// IndraMotionMlc1/Application/CheckBounds
(*
General Header
----------------------------------------------------------------------------------------------
Short description      : Function to check access to array within valid bounds.
                         After inserting/removing this function, no online-change will be possible! A complete download will be necessary!
Version                : 14.1.0.0
Author                 : DC-IA/EAM3 (MD)
Date                   : 2015-01-12
Company                : Bosch Rexroth AG
Target                 : IndraLogic XLC/MLC
Functional description : This function will be called implicitly before the read/write access
                         to arrays takes places.
                         The index of the subsequent array accesses is checked for valid
                         limits.
                         In case of invalid access, an error is entered in the diagnostic
                         logbook and the application is stopped due to an access violation to
                         avoid machine damage.
                         In this case, check the callstack (menu Debug/Callstack) and modify
                         the faulty logic. 
Handling specials      : This function increases the cycle time of all IEC-tasks using array
                         accesses. 
                         The increase depends on the number of the read/write accesses to
                         arrays.
                         After inserting/removing this function, no online-change will be possible! 
                         A complete download will be necessary!
						 This is an exemplary implementation of the function. 
                         The implementation has to be adjusted to your application/machine.
						 Per default, the PLC-Task will generate an access violation which leads to
                         an application stop and a F5-error with error reaction respectively.
                         Please verify whether this default behaviour can damage your machine 
                         or lead to a complex recommissioning. 
                         In this case, adapt the error reaction to your application.
						 
                         If your application isn't too time-critical, you should leave this function 
						 while commissioning the machine and production in your application.  
                         If you remove this funciton, ensure that your code is faultless.
                         
                         Do not modify the declaration of this function! 
                         Do not change the attributes above the function header!
----------------------------------------------------------------------------------------------
*)
{attribute 'check_bounds'}
{attribute 'no_check'}
{attribute 'signature_flag' := '1073741824'}
FUNCTION CheckBounds : DINT
VAR_INPUT
	index, lower, upper: DINT;
END_VAR
VAR
	{attribute 'hide'}
	bByte: BYTE;
	ptNull: POINTER TO BYTE :=0;
	errstr: STRING;
	
END_VAR

(*************************************************************
This function was generated by the 'check array access'
option of the controllers 'properties' dialog box.
If you delete this comment, the 'check array access' option
of the controllers 'properties' dialog box will be removed.
**************************************************************)
    (**************************************************************************************************)
    (* The implementation has to be adjusted to your application/machine.                             *)
    (* This is an exemplary implementation of the function.                                           *)
    (* Per default, an access violation is generated to avoid machine damage                          *)
    (* Check the Call Stack (menu Debug/Callstack) and modify the faulty logic!                       *)
    (**************************************************************************************************)

IF  index < lower THEN 
	errstr:= 'CheckBounds: Lower arrayindex ';
	errstr:=CONCAT(STR1:=errstr  , STR2:= DINT_TO_STRING(lower));
	errstr:=CONCAT(STR1:=errstr  , STR2:= ' underrunned by ');
	errstr:=CONCAT(STR1:=errstr  , STR2:= DINT_TO_STRING(index));
//  This pragma may be removed: 
	{info 'CheckBounds: Please implement your own error reaction below'}
//  EXAMPLE 1 (default): 
//  Set a F0-Error into the diagnostic- and error memory
//  Triggering an access violation --> Application will be stopped and leads to a F5-Error

  ML_SetDiagEntry(
	Severity:= E_LOG_SEVERITY.ERROR, 
	Class:= E_LOG_CLASS.CLASS_0, 
	Facility:= E_LOG_FACILITY.USER, 
	Code:= 0, 
	Text:= ADR(errstr));

	bByte:=ptNull^;(*triggering an access violation *)

// EXAMPLE 2:
// Limit the faulty index to the lower index 
//     -> no memory will be overwritten
//     -> Keep PLC-task and motion running
// Set a E0-Warning into the diagnostic- and error memory
// NOTE: There is still an implementation error in your application code!

//  ML_SetDiagEntry(
//	Severity:= E_LOG_SEVERITY.WARNING, 
//	Class:= E_LOG_CLASS.CLASS_0, 
//	Facility:= E_LOG_FACILITY.USER, 
//	Code:= 0, 
//	Text:= ADR(errstr));
// 
//	CheckBounds := lower; //access to the lower index only 
//  return;
	
ELSIF  index > upper THEN
	errstr:= 'CheckBounds: Higher arrayindex ';
	errstr:=CONCAT(STR1:=errstr  , STR2:= DINT_TO_STRING(upper));
	errstr:=CONCAT(STR1:=errstr  , STR2:= ' overrunned by ');
	errstr:=CONCAT(STR1:=errstr  , STR2:= DINT_TO_STRING(index));

//  this pragma may be removed: 
	{info 'CheckBounds: Please implement your own error reaction below'}
//  example 1 (default): 
//  set a F0-Error into the diagnostic- and error memory
//  triggering an access violation --> Application will be stopped and leads to a F5-Error

  ML_SetDiagEntry(
	Severity:= E_LOG_SEVERITY.ERROR, 
	Class:= E_LOG_CLASS.CLASS_0, 
	Facility:= E_LOG_FACILITY.USER, 
	Code:= 0, 
	Text:= ADR(errstr));

	bByte:=ptNull^;(*triggering an access violation *)

//example 2:
// Limit the faulty index to the upper index 
//     -> no memory will be overwritten
//     -> Keep PLC-task and motion running
// Set a E0-Warning into the diagnostic- and error memory
// NOTE: There is still an implementation error in your application code!

//  ML_SetDiagEntry(
//	Severity:= E_LOG_SEVERITY.WARNING, 
//	Class:= E_LOG_CLASS.CLASS_0, 
//	Facility:= E_LOG_FACILITY.USER, 
//	Code:= 0, 
//	Text:= ADR(errstr));
// 
//	CheckBounds := upper; //access to the upper index only 
//  return;

ELSE // access to array is ok  
	CheckBounds := index;
END_IF

END_FUNCTION

// IndraMotionMlc1/Application/POUs/Useless/MotionProg
PROGRAM MotionProg
VAR
	b_enable_1: BOOL;
	MC_Power_0: MC_POWER;
	b_enable_on_1: BOOL;
	b_move_1: BOOL;
	MC_MoveVelocity_0: MC_MoveVelocity;
	vel: REAL;
	b_enable_2: BOOL;
	MC_Power_1: MC_POWER;
	b_enable_on_2: BOOL;
	b_move_2: BOOL;
	MC_MoveVelocity_1: MC_MoveVelocity;
	b_enable_3: BOOL;
	MC_Power_2: MC_POWER;
	b_enable_on_3: BOOL;
	b_move_3: BOOL;
	MC_MoveVelocity_2: MC_MoveVelocity;
	b_power: BOOL;
	b_vel_az1: BOOL;
	b_enable_az1: BOOL;
	b_enable_az2: BOOL;
	b_torque_az2: BOOL;
	b_torque_on_2: BOOL;
	MC_torque_az2: MC_TorqueControl;
	b_enable_el_1: BOOL;
	b_move_el_1: BOOL;
	b_torque_az1: BOOL;
	MC_torque_az1: MC_TorqueControl;
	b_torque_on_1: BOOL;
	b_vel_2: BOOL;
END_VAR

motionprog.P_MOTION();

ACTION P_MOTION:
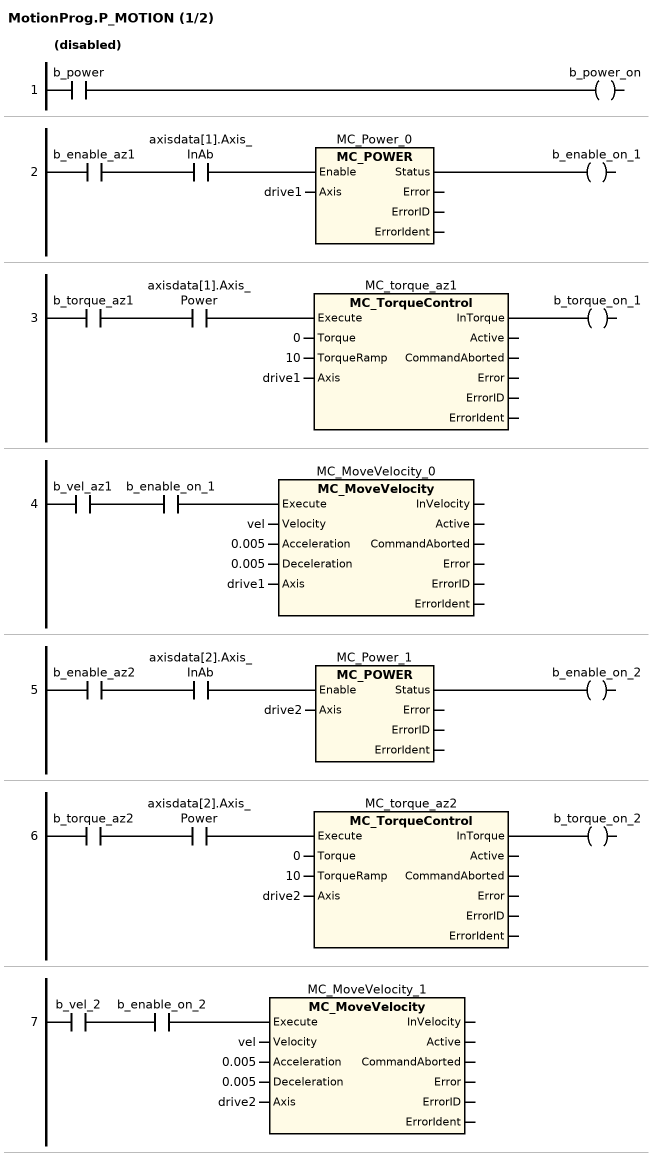
// NETWORK 1 (disabled)
// b_power_on := b_power;

// NETWORK 2
MC_Power_0(Enable := b_enable_az1 AND axisdata[1].Axis_InAb, Axis := drive1); // MC_POWER
b_enable_on_1 := MC_Power_0.Status;

// NETWORK 3
MC_torque_az1(
    Execute := b_torque_az1 AND axisdata[1].Axis_Power,
    Torque := 0,
    TorqueRamp := 10,
    Axis := drive1); // MC_TorqueControl
b_torque_on_1 := MC_torque_az1.InTorque;

// NETWORK 4
MC_MoveVelocity_0(
    Execute := b_vel_az1 AND b_enable_on_1,
    Velocity := vel,
    Acceleration := 0.005,
    Deceleration := 0.005,
    Axis := drive1); // MC_MoveVelocity

// NETWORK 5
MC_Power_1(Enable := b_enable_az2 AND axisdata[2].Axis_InAb, Axis := drive2); // MC_POWER
b_enable_on_2 := MC_Power_1.Status;

// NETWORK 6
MC_torque_az2(
    Execute := b_torque_az2 AND axisdata[2].Axis_Power,
    Torque := 0,
    TorqueRamp := 10,
    Axis := drive2); // MC_TorqueControl
b_torque_on_2 := MC_torque_az2.InTorque;

// NETWORK 7
MC_MoveVelocity_1(
    Execute := b_vel_2 AND b_enable_on_2,
    Velocity := vel,
    Acceleration := 0.005,
    Deceleration := 0.005,
    Axis := drive2); // MC_MoveVelocity

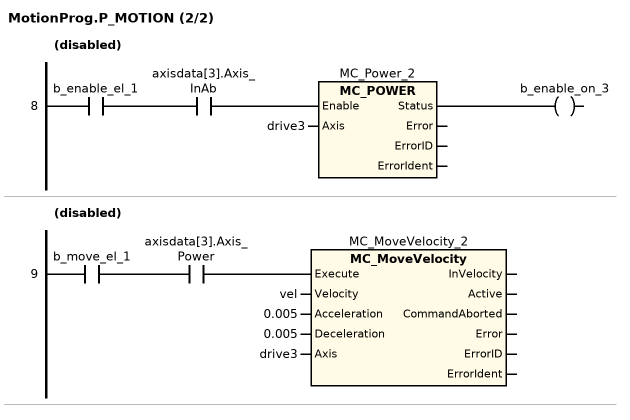
// NETWORK 8 (disabled)
// MC_Power_2(Enable := b_enable_el_1 AND axisdata[3].Axis_InAb, Axis := drive3); // MC_POWER
// b_enable_on_3 := MC_Power_2.Status;

// NETWORK 9 (disabled)
// MC_MoveVelocity_2(
//     Execute := b_move_el_1 AND axisdata[3].Axis_Power,
//     Velocity := vel,
//     Acceleration := 0.005,
//     Deceleration := 0.005,
//     Axis := drive3); // MC_MoveVelocity
END_ACTION

END_PROGRAM

// IndraMotionMlc1/Application/POUs/Panel Function/P_LED
(*
This progrom is bulit for lighting the led in the panelbox which describe the limit.
1)If the angle is reach the limit value,we use the Function Block MB_WriteParameter to setting 
special value to the parameter FP_P_0_0304 of the relative drive.so that the led will be lighted.
2)Besides,when the position of azimuth axis is at the zone,60 degrees nearby the limit,the led of azimuth will flicker every 2 seconds.
Similar with azimuth,the elevation LED will flicker at the 5-degrees-zone nearby limit,and the FeedIndexer LED will flicker at the 30-degrees-zone nearby limit.
*)
PROGRAM P_LED
VAR
(*the definition of Blink function blocks*)
	fb_blink_LED_az: BLINK;
	fb_blink_write_az: BLINK;
	fb_blink_LED_el: BLINK;
	fb_blink_write_el: BLINK;
	fb_blink_LED_FI: BLINK;
	fb_blink_write_FI: BLINK;
	t_LED_az: TIME;
	t_LED_el: TIME;
	t_LED_FI: TIME;
	b_LED_az: BOOL;
	b_LED_el: BOOL;
	b_LED_FI: BOOL;
(*the definition of function blocks for Writing p304 Parameter*)
	fb_write_p304_d2: MB_WriteParameter;(*the I/O of azimuth LED is on drive2*)
	fb_write_p304_d4: MB_WriteParameter;(*the I/O of elevation LED is on drive4*)
	fb_write_p304_d5: MB_WriteParameter;(*the I/O of FeedIndexer LED is on drive5*)
(*when the P304 parameter equal to 512,only the 9th on the I/O is set;
when the P304 parameter equal to 1024,only the 10th on the I/O is set;
when the P304 parameter equal to 0,all the I/O is reset;*)
	i_p304_az: INT;
	i_p304_el: INT;
	i_p304_FI: INT;
END_VAR

IF b_local_on=TRUE THEN
	b_local_led:=TRUE;
ELSE
	b_local_led:=FALSE;
END_IF

IF b_remote_on=TRUE THEN
	b_remote_led:=TRUE;
ELSE
	b_remote_led:=FALSE;
END_IF

IF b_ESTOP_door=TRUE THEN
	b_estop_led :=TRUE;
ELSE
	b_estop_led :=FALSE;
END_IF

   IF master_status.4 =FALSE THEN
	   b_normal_led:=TRUE;
	   b_error_led:=FALSE;
   ELSE
   	   b_normal_led:=FALSE;
	   b_error_led:=TRUE;
   END_IF


(*
IF b_local_on=TRUE THEN
(*<<<<<<<<<<<<<<<<<<<<<<<<<<<<<<<<LED Of azimuth>>>>>>>>>>>>>>>>>>>>>>>>>>>>>>>>>*)
	IF r_pos_az>=0 AND r_pos_az<=180 THEN
		i_p304_az:=0;
	ELSIF r_pos_az>180 AND r_pos_az<358.5 THEN
		t_LED_az:=T#2.2s;
		IF b_LED_az= TRUE THEN
			i_p304_az:=0;
		ELSE
			i_p304_az:=512;
		END_IF
	ELSIF r_pos_az>=358.5 THEN
		i_p304_az:=512;
	ELSIF r_pos_az<0 AND r_pos_az>-178.5 THEN
		t_LED_az:=T#2.2s;
		IF b_LED_az= TRUE THEN
			i_p304_az:=0;
		ELSE
			i_p304_az:=1024;
		END_IF
	ELSIF r_pos_az<=-178.5 THEN
		i_p304_az:=1024;
	END_IF
(*<<<<<<<<<<<<<<<<<<<<<<<<<<<<<<<<LED Of elevation>>>>>>>>>>>>>>>>>>>>>>>>>>>>>>>>>*)
	IF r_pos_el>=25 AND r_pos_el<=80 THEN
		i_p304_el:=0;
	ELSIF r_pos_el>80 AND r_pos_el<=90.1 THEN
		t_LED_el:=T#2.2s;
		IF b_LED_el= TRUE THEN
			i_p304_el:=0;
		ELSE
			i_p304_el:=512;
		END_IF
	ELSIF r_pos_el>90.1 THEN
		i_p304_el:=512;
	ELSIF r_pos_el>25 AND r_pos_el<=15 THEN
		t_LED_el:=T#2.2s;
		IF b_LED_el= TRUE THEN
			i_p304_el:=0;
		ELSE
			i_p304_el:=1024;
		END_IF
	ELSIF r_pos_el<15 THEN
		i_p304_el:=1024;
	END_IF
(*<<<<<<<<<<<<<<<<<<<<<<<<<<<<<<<<LED Of FeedIndexer>>>>>>>>>>>>>>>>>>>>>>>>>>>>>>>>>*)
	IF r_pos_FI>=-120 AND r_pos_FI<=120 THEN
		i_p304_FI:=0;
	ELSIF r_pos_FI>120 AND r_pos_FI<=178.5 THEN
		t_LED_FI:=T#2.2s;
		IF b_LED_FI= TRUE THEN
			i_p304_FI:=0;
		ELSE
			i_p304_FI:=512;
		END_IF
	ELSIF r_pos_FI>178.5 THEN
		i_p304_FI:=512;
	ELSIF r_pos_FI<-120 AND r_pos_FI>=-178.5 THEN
		t_LED_FI:=T#2.2s;
		IF b_LED_FI= TRUE THEN
			i_p304_FI:=0;
		ELSE
			i_p304_FI:=1024;
		END_IF
	ELSIF r_pos_FI<-178.5 THEN
		i_p304_FI:=1024;
	END_IF
ELSE
(*if not at local situation,the LED is dark*)
(*For testing LED,write i_p304_az:=1536;i_p304_el:=1536;i_p304_FI:=1536;*)
	i_p304_az:=0;
	i_p304_el:=0;
	i_p304_FI:=0;
END_IF

(*transfer the sub-program A_w_P304 to white value to the parameter FP_P_0_0304*)
P_LED.A_w_P304;*)

ACTION A_w_P304:
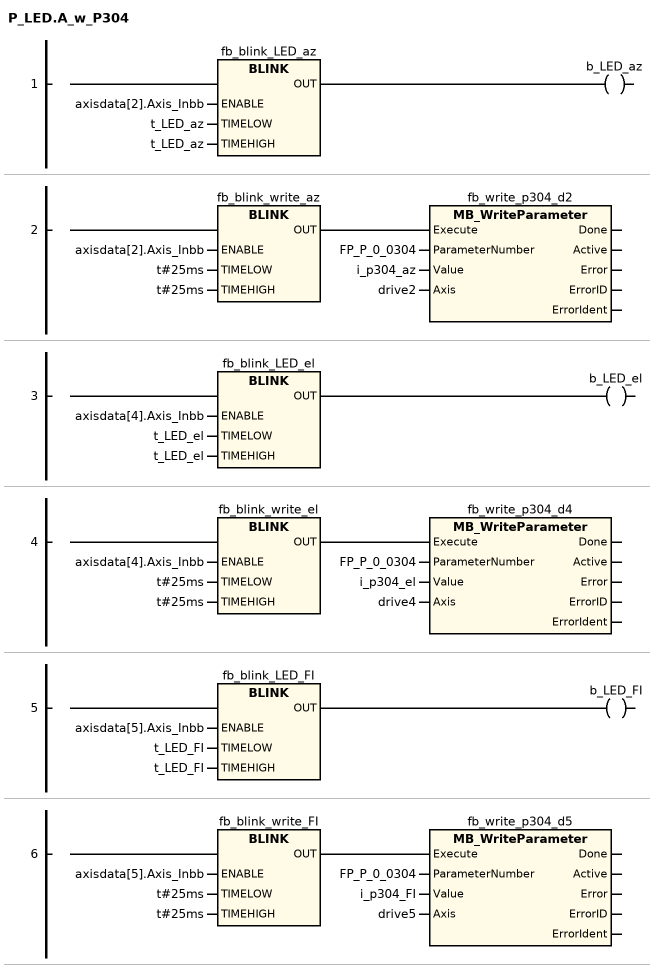
// NETWORK 1
fb_blink_LED_az(ENABLE := axisdata[2].Axis_Inbb, TIMELOW := t_LED_az, TIMEHIGH := t_LED_az); // BLINK
b_LED_az := fb_blink_LED_az.OUT;

// NETWORK 2
fb_blink_write_az(ENABLE := axisdata[2].Axis_Inbb, TIMELOW := t#25ms, TIMEHIGH := t#25ms); // BLINK
fb_write_p304_d2(
    Execute := fb_blink_write_az.OUT,
    ParameterNumber := FP_P_0_0304,
    Value := i_p304_az,
    Axis := drive2); // MB_WriteParameter

// NETWORK 3
fb_blink_LED_el(ENABLE := axisdata[4].Axis_Inbb, TIMELOW := t_LED_el, TIMEHIGH := t_LED_el); // BLINK
b_LED_el := fb_blink_LED_el.OUT;

// NETWORK 4
fb_blink_write_el(ENABLE := axisdata[4].Axis_Inbb, TIMELOW := t#25ms, TIMEHIGH := t#25ms); // BLINK
fb_write_p304_d4(
    Execute := fb_blink_write_el.OUT,
    ParameterNumber := FP_P_0_0304,
    Value := i_p304_el,
    Axis := drive4); // MB_WriteParameter

// NETWORK 5
fb_blink_LED_FI(ENABLE := axisdata[5].Axis_Inbb, TIMELOW := t_LED_FI, TIMEHIGH := t_LED_FI); // BLINK
b_LED_FI := fb_blink_LED_FI.OUT;

// NETWORK 6
fb_blink_write_FI(ENABLE := axisdata[5].Axis_Inbb, TIMELOW := t#25ms, TIMEHIGH := t#25ms); // BLINK
fb_write_p304_d5(
    Execute := fb_blink_write_FI.OUT,
    ParameterNumber := FP_P_0_0304,
    Value := i_p304_FI,
    Axis := drive5); // MB_WriteParameter
END_ACTION

END_PROGRAM

// IndraMotionMlc1/Application/POUs/Panel Function/P_Lock_Panel_TCP
(*This program is bulit for lock the antenna for stow and maintain,and for unlock the antenna.
It mainly contains goto function,the control of AC moter,and the protect for safety*)
PROGRAM P_Lock_Panel_TCP
VAR

(*<<<<<<<<<<<<<<<<<<<the allow for the lock moter>>>>>>>>>>>>>>>>>*)
	b_lock_allow_0: BOOL;
	b_lock_allow_20: BOOL;
(*the definition of rise trigger,The function block R_TRIG detects a rising edge. *)
	rtrig_lock_stow: R_TRIG;
	rtrig_lock_maintain: R_TRIG;
	rtrig_reset_TCP_unlock: R_TRIG;
	rtrig_reset_TCP_lock: R_TRIG;
	rtrig_enable_unlock: R_TRIG;
(*The function block Timer On Delay implements a turn-on delay*)
	ton_stow_0: TON;
	ton_maintain_20: TON;
	ton_reset_lock: TON;
	ton_reset_unlock: TON;
(*the fixed position according to the hole*)
	r_postion_stow: REAL;
	r_position_maintain: REAL;
(*move the elevation to the fixed position*)
	fb_move_AZ_0: MC_MoveAbsolute;
	fb_move_el_20: MC_MoveAbsolute;
	fb_self_reset_stow: R_TRIG;
	fb_ton_self_reset_stow: TON;
	b_lock_allow_21: BOOL;
	fb_self_reset_maintain: R_TRIG;
	fb_ton_self_reset_maintain: TON;
	b_off_stow: R_TRIG;
	b_off_maintain: R_TRIG;
	fb_move_EL_0: MC_MoveAbsolute;
END_VAR

(*<<<<<<<<<<<<<<<<<<<<write the stow and maintain position according to IP>>>>>>>>>>>>>>>>>>>>>>>>>>>>>>>>>>>>*)
(*every antenna maybe has the different stow position and maintain position from the others*)
str_1xx:=RIGHT(str_MLC_ip,3);(*for get the last 3 number of IP in MLC*)
IF str_1xx='101' THEN
	r_postion_stow:=0;
	r_position_maintain:=20.15;
ELSIF str_1xx='102' THEN
	r_postion_stow:=0;
	r_position_maintain:=20.820;
ELSIF str_1xx='103' THEN
	r_postion_stow:=0;
	r_position_maintain:=20.950;
ELSIF str_1xx='104' THEN
	r_postion_stow:=0;
	r_position_maintain:=20.9;
ELSIF str_1xx='105' THEN
	r_postion_stow:=0;
	r_position_maintain:=20.930;
ELSIF str_1xx='106' THEN
	r_postion_stow:=0;
	r_position_maintain:=20.800;
ELSIF str_1xx='107' THEN
	r_postion_stow:=90.00;
	r_position_maintain:=20.850;
ELSIF str_1xx='108' THEN
	r_postion_stow:=90.00;
	r_position_maintain:=21.100;
ELSIF str_1xx='109' THEN
	r_postion_stow:=90.00;
	r_position_maintain:=21.000;
ELSIF str_1xx='110' THEN
	r_postion_stow:=0;
	r_position_maintain:=21.000;
ELSIF str_1xx='111' THEN
	r_postion_stow:=0;
	r_position_maintain:=21.000;
ELSIF str_1xx='112' THEN
	r_postion_stow:=0;
	r_position_maintain:=21.100;
ELSIF str_1xx='113' THEN
	r_postion_stow:=0;
	r_position_maintain:=21.000;
ELSIF str_1xx='114' THEN
	r_postion_stow:=0;
	r_position_maintain:=21.000;
ELSIF str_1xx='115' THEN
	r_postion_stow:=0;
	r_position_maintain:=21.000;
ELSIF str_1xx='116' THEN
	r_postion_stow:=0;
	r_position_maintain:=21.000;
ELSIF str_1xx='117' THEN
	r_postion_stow:=0;
	r_position_maintain:=21.000;
ELSIF str_1xx='118' THEN
	r_postion_stow:=0;
	r_position_maintain:=20.950;
ELSIF str_1xx='119' THEN
	r_postion_stow:=0;
	r_position_maintain:=20.950;
ELSIF str_1xx='120' THEN
	r_postion_stow:=0;
	r_position_maintain:=21.000;
ELSIF str_1xx='121' THEN
	r_postion_stow:=0;
	r_position_maintain:=21.000;
ELSIF str_1xx='122' THEN
	r_postion_stow:=0;
	r_position_maintain:=21.000;
ELSIF str_1xx='123' THEN
	r_postion_stow:=0;
	r_position_maintain:=21.000;
ELSIF str_1xx='124' THEN
	r_postion_stow:=0;
	r_position_maintain:=21.000;
ELSIF str_1xx='125' THEN
	r_postion_stow:=0;
	r_position_maintain:=21.000;
ELSIF str_1xx='126' THEN
	r_postion_stow:=0;
	r_position_maintain:=21.000;
ELSIF str_1xx='127' THEN
	r_postion_stow:=0;
	r_position_maintain:=21.000;
ELSIF str_1xx='128' THEN
	r_postion_stow:=0;
	r_position_maintain:=21.000;
ELSIF str_1xx='129' THEN
	r_postion_stow:=0;
	r_position_maintain:=21.000;
ELSIF str_1xx='130' THEN
	r_postion_stow:=0;
	r_position_maintain:=20.950;
ELSIF str_1xx='131' THEN
	r_postion_stow:=0;
	r_position_maintain:=21.000;
ELSIF str_1xx='132' THEN
	r_postion_stow:=0;
	r_position_maintain:=21.000;
ELSIF str_1xx='133' THEN
	r_postion_stow:=0;
	r_position_maintain:=21.000;
ELSIF str_1xx='134' THEN
	r_postion_stow:=0;
	r_position_maintain:=21.000;
ELSIF str_1xx='135' THEN
	r_postion_stow:=0.00;
	r_position_maintain:=21.000;
ELSIF str_1xx='136' THEN
	r_postion_stow:=0.00;
	r_position_maintain:=21.000;

(*test*)
ELSIF str_1xx='1.1' THEN
	r_postion_stow:=0.00;
	r_position_maintain:=20.9;
ELSE
	r_postion_stow:=0;
	r_position_maintain:=11;
END_IF
(*<<<<<<<<<<<<<<<<<<<<<<<<<<<<<<<<if the elevation position is nearby the fixed value,then allow the lock action>>>>>>>>>>>>>>>>>>>>>>>>>>>>>>>>>>>>>>>>>>>>>>>>>>>*)
IF ABS(axisdata[1].rActualPosition_i-0)<0.01 THEN
	b_lock_allow_0:=TRUE;
ELSE
	b_lock_allow_0:=FALSE;
END_IF

IF b_stow_pin_limit_lock = FALSE AND ABS(axisdata[1].rActualPosition_i-r_postion_stow)< 0.1 THEN
	b_stow_lock:=TRUE;
ELSE
	b_stow_lock:=FALSE;
END_IF;

P_Lock_Panel_TCP.A_LOCK();

ACTION A_LOCK:
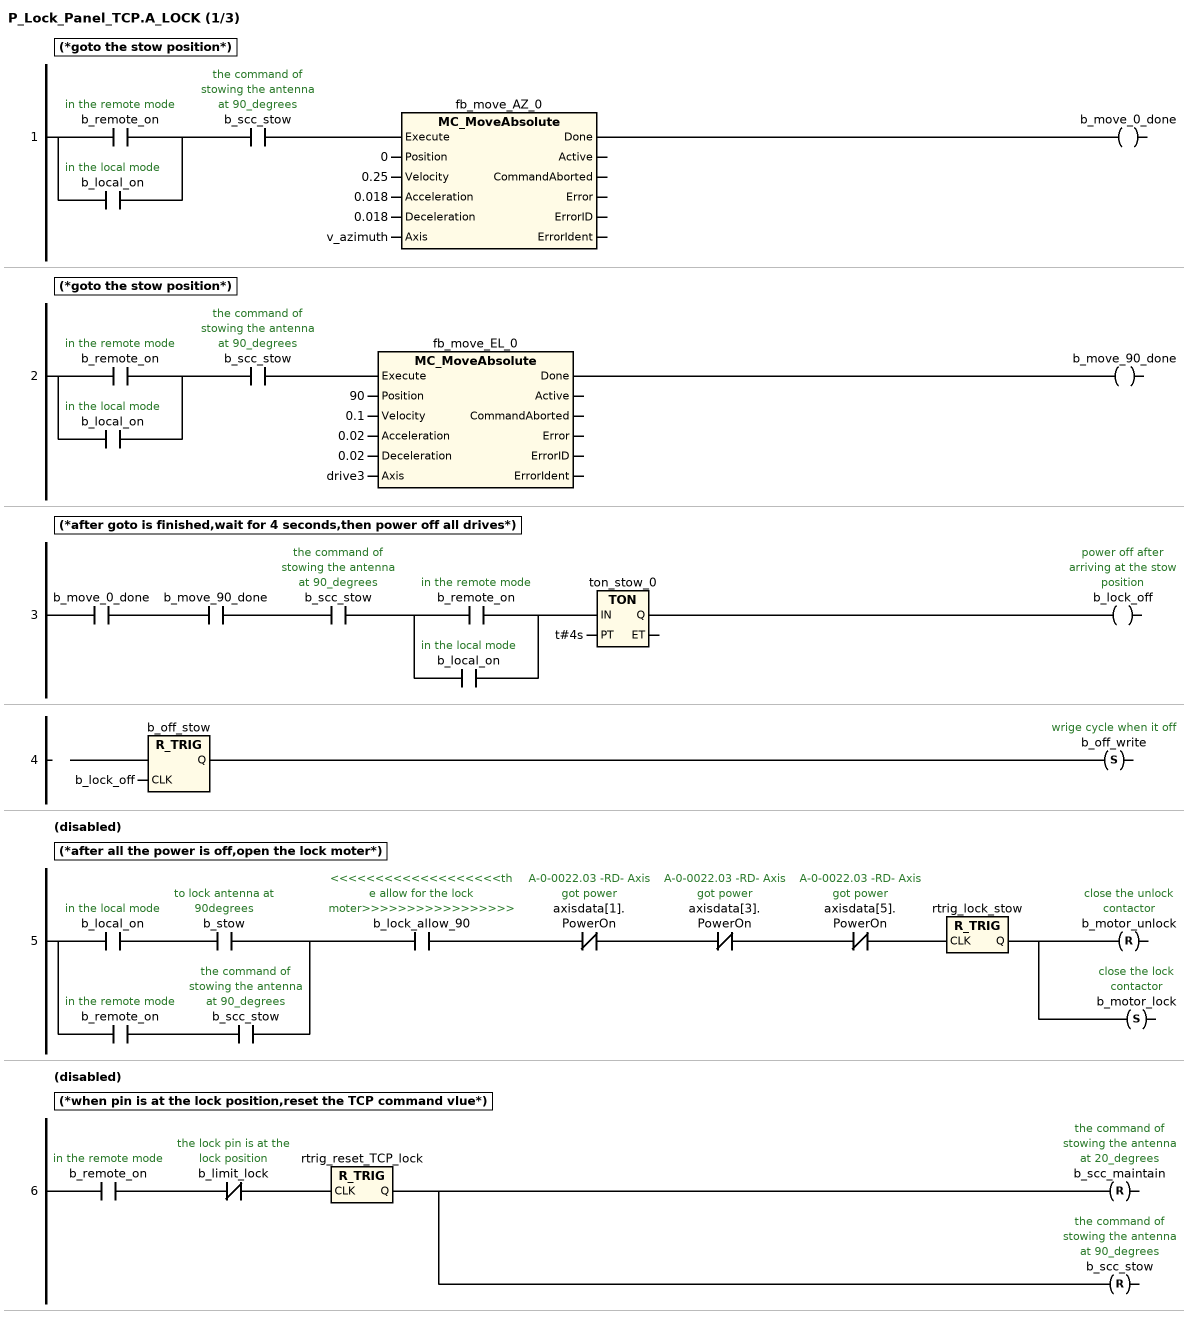
// NETWORK 1
//   fb_move_AZ_0: move the elevation to the fixed position
//   b_remote_on: in the remote mode
//   b_local_on: in the local mode
//   b_scc_stow: the command of stowing the antenna at 90_degrees
//   v_azimuth: Virtual axis "v_elevation" with axis number 8
// label: (*goto the stow position*)
fb_move_AZ_0(
    Execute := (b_remote_on OR b_local_on) AND b_scc_stow,
    Position := 0,
    Velocity := 0.25,
    Acceleration := 0.018,
    Deceleration := 0.018,
    Axis := v_azimuth); // MC_MoveAbsolute
b_move_0_done := fb_move_AZ_0.Done;

// NETWORK 2
//   fb_move_EL_0: move the elevation to the fixed position
//   b_remote_on: in the remote mode
//   b_local_on: in the local mode
//   b_scc_stow: the command of stowing the antenna at 90_degrees
//   drive3: Virtual axis "v_elevation" with axis number 8
// label: (*goto the stow position*)
fb_move_EL_0(
    Execute := (b_remote_on OR b_local_on) AND b_scc_stow,
    Position := 90,
    Velocity := 0.1,
    Acceleration := 0.02,
    Deceleration := 0.02,
    Axis := drive3); // MC_MoveAbsolute
b_move_90_done := fb_move_EL_0.Done;

// NETWORK 3
//   ton_stow_0: The function block Timer On Delay implements a turn-on delay
//   b_scc_stow: the command of stowing the antenna at 90_degrees
//   b_remote_on: in the remote mode
//   b_local_on: in the local mode
//   b_lock_off: power off after arriving at the stow position
// label: (*after goto is finished,wait for 4 seconds,then power off all drives*)
ton_stow_0(IN := b_move_0_done AND b_move_90_done AND b_scc_stow AND (b_remote_on OR b_local_on), PT := t#4s); // TON
b_lock_off := ton_stow_0.Q;

// NETWORK 4
//   b_lock_off: power off after arriving at the stow position
//   b_off_write: wrige cycle when it off
b_off_stow(CLK := b_lock_off); // R_TRIG
b_off_write S= b_off_stow.Q;

// NETWORK 5 (disabled)
//   rtrig_lock_stow: the definition of rise trigger,The function block R_TRIG detects a rising edge.
//   b_local_on: in the local mode
//   b_stow: to lock antenna at 90degrees
//   b_remote_on: in the remote mode
//   b_scc_stow: the command of stowing the antenna at 90_degrees
//   b_lock_allow_90: <<<<<<<<<<<<<<<<<<<the allow for the lock moter>>>>>>>>>>>>>>>>>
//   axisdata[1].PowerOn: A-0-0022.03 -RD- Axis got power
//   axisdata[3].PowerOn: A-0-0022.03 -RD- Axis got power
//   axisdata[5].PowerOn: A-0-0022.03 -RD- Axis got power
//   b_motor_unlock: close the unlock contactor
//   b_motor_lock: close the lock contactor
// label: (*after all the power is off,open the lock moter*)
// rtrig_lock_stow(CLK := (b_local_on AND b_stow OR b_remote_on AND b_scc_stow) AND b_lock_allow_90 AND NOT axisdata[1].PowerOn AND NOT axisdata[3].PowerOn AND NOT axisdata[5].PowerOn); // R_TRIG
// b_motor_unlock R= rtrig_lock_stow.Q;
// b_motor_lock S= rtrig_lock_stow.Q;

// NETWORK 6 (disabled)
//   b_remote_on: in the remote mode
//   b_limit_lock: the lock pin is at the lock position
//   b_scc_maintain: the command of stowing the antenna at 20_degrees
//   b_scc_stow: the command of stowing the antenna at 90_degrees
// label: (*when pin is at the lock position,reset the TCP command vlue*)
// rtrig_reset_TCP_lock(CLK := b_remote_on AND NOT b_limit_lock); // R_TRIG
// b_scc_maintain R= rtrig_reset_TCP_lock.Q;
// b_scc_stow R= rtrig_reset_TCP_lock.Q;

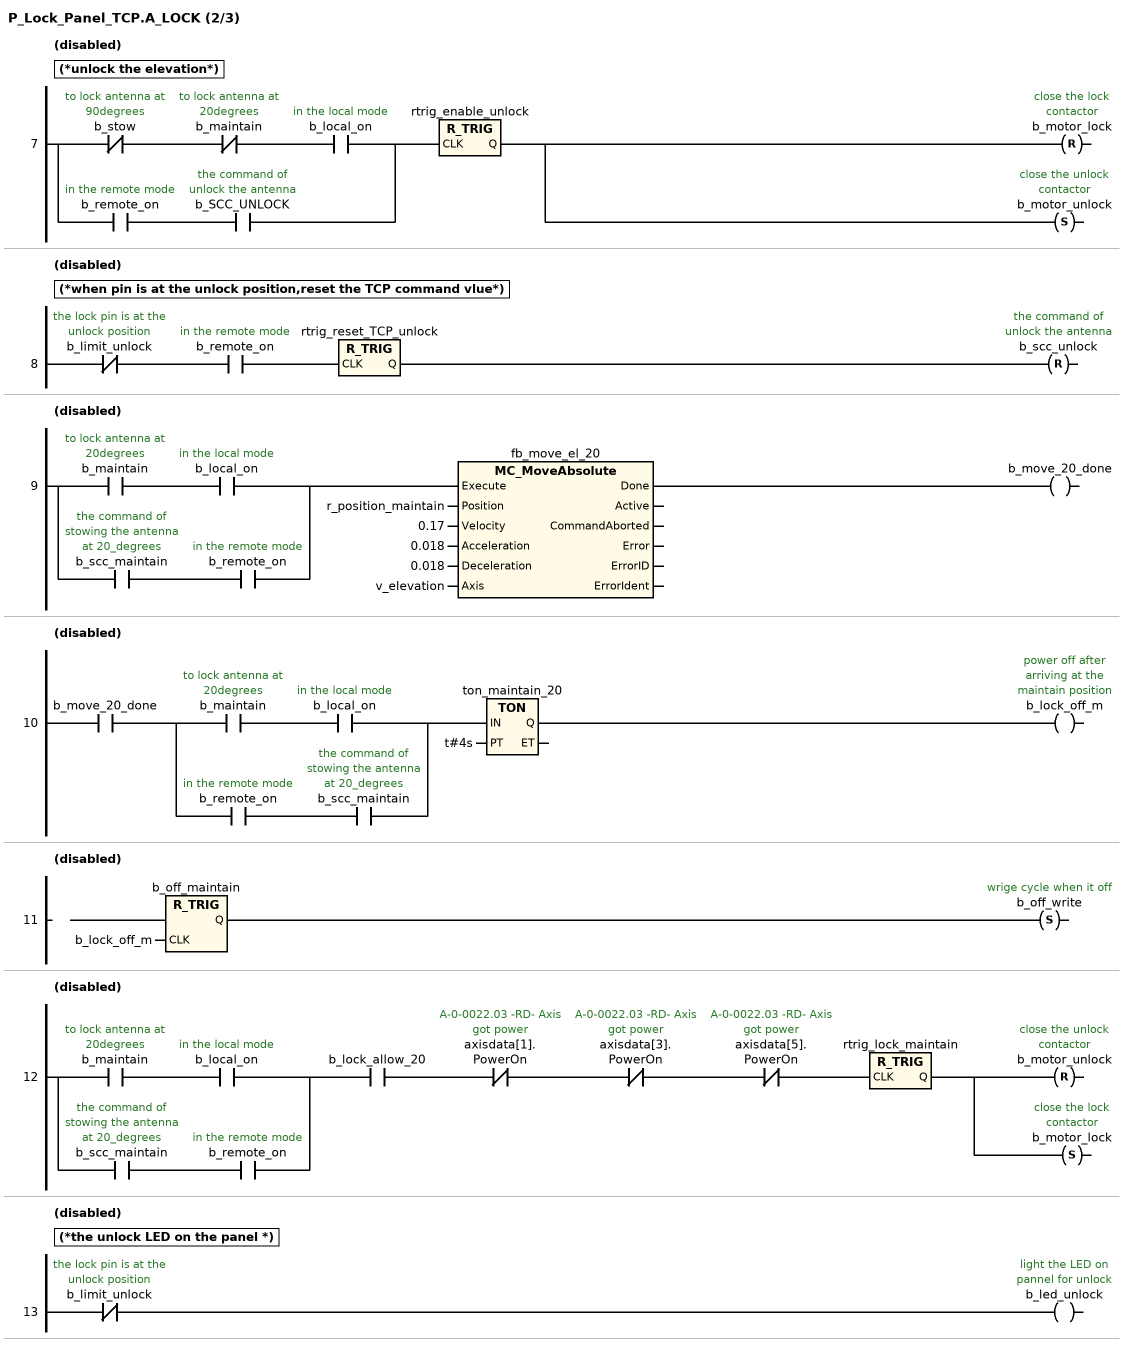
// NETWORK 7 (disabled)
//   b_stow: to lock antenna at 90degrees
//   b_maintain: to lock antenna at 20degrees
//   b_local_on: in the local mode
//   b_remote_on: in the remote mode
//   b_SCC_UNLOCK: the command of unlock the antenna
//   b_motor_lock: close the lock contactor
//   b_motor_unlock: close the unlock contactor
// label: (*unlock the elevation*)
// rtrig_enable_unlock(CLK := NOT b_stow AND NOT b_maintain AND b_local_on OR b_remote_on AND b_SCC_UNLOCK); // R_TRIG
// b_motor_lock R= rtrig_enable_unlock.Q;
// b_motor_unlock S= rtrig_enable_unlock.Q;

// NETWORK 8 (disabled)
//   b_limit_unlock: the lock pin is at the unlock position
//   b_remote_on: in the remote mode
//   b_scc_unlock: the command of unlock the antenna
// label: (*when pin is at the unlock position,reset the TCP command vlue*)
// rtrig_reset_TCP_unlock(CLK := NOT b_limit_unlock AND b_remote_on); // R_TRIG
// b_scc_unlock R= rtrig_reset_TCP_unlock.Q;

// NETWORK 9 (disabled)
//   b_maintain: to lock antenna at 20degrees
//   b_local_on: in the local mode
//   b_scc_maintain: the command of stowing the antenna at 20_degrees
//   b_remote_on: in the remote mode
//   v_elevation: Virtual axis "v_elevation" with axis number 8
// fb_move_el_20(
//     Execute := b_maintain AND b_local_on OR b_scc_maintain AND b_remote_on,
//     Position := r_position_maintain,
//     Velocity := 0.17,
//     Acceleration := 0.018,
//     Deceleration := 0.018,
//     Axis := v_elevation); // MC_MoveAbsolute
// b_move_20_done := fb_move_el_20.Done;

// NETWORK 10 (disabled)
//   b_maintain: to lock antenna at 20degrees
//   b_local_on: in the local mode
//   b_remote_on: in the remote mode
//   b_scc_maintain: the command of stowing the antenna at 20_degrees
//   b_lock_off_m: power off after arriving at the maintain position
// ton_maintain_20(IN := b_move_20_done AND (b_maintain AND b_local_on OR b_remote_on AND b_scc_maintain), PT := t#4s); // TON
// b_lock_off_m := ton_maintain_20.Q;

// NETWORK 11 (disabled)
//   b_lock_off_m: power off after arriving at the maintain position
//   b_off_write: wrige cycle when it off
// b_off_maintain(CLK := b_lock_off_m); // R_TRIG
// b_off_write S= b_off_maintain.Q;

// NETWORK 12 (disabled)
//   b_maintain: to lock antenna at 20degrees
//   b_local_on: in the local mode
//   b_scc_maintain: the command of stowing the antenna at 20_degrees
//   b_remote_on: in the remote mode
//   axisdata[1].PowerOn: A-0-0022.03 -RD- Axis got power
//   axisdata[3].PowerOn: A-0-0022.03 -RD- Axis got power
//   axisdata[5].PowerOn: A-0-0022.03 -RD- Axis got power
//   b_motor_unlock: close the unlock contactor
//   b_motor_lock: close the lock contactor
// rtrig_lock_maintain(CLK := (b_maintain AND b_local_on OR b_scc_maintain AND b_remote_on) AND b_lock_allow_20 AND NOT axisdata[1].PowerOn AND NOT axisdata[3].PowerOn AND NOT axisdata[5].PowerOn); // R_TRIG
// b_motor_unlock R= rtrig_lock_maintain.Q;
// b_motor_lock S= rtrig_lock_maintain.Q;

// NETWORK 13 (disabled)
//   b_limit_unlock: the lock pin is at the unlock position
//   b_led_unlock: light the LED on pannel for unlock
// label: (*the unlock LED on the panel *)
// b_led_unlock := NOT b_limit_unlock;

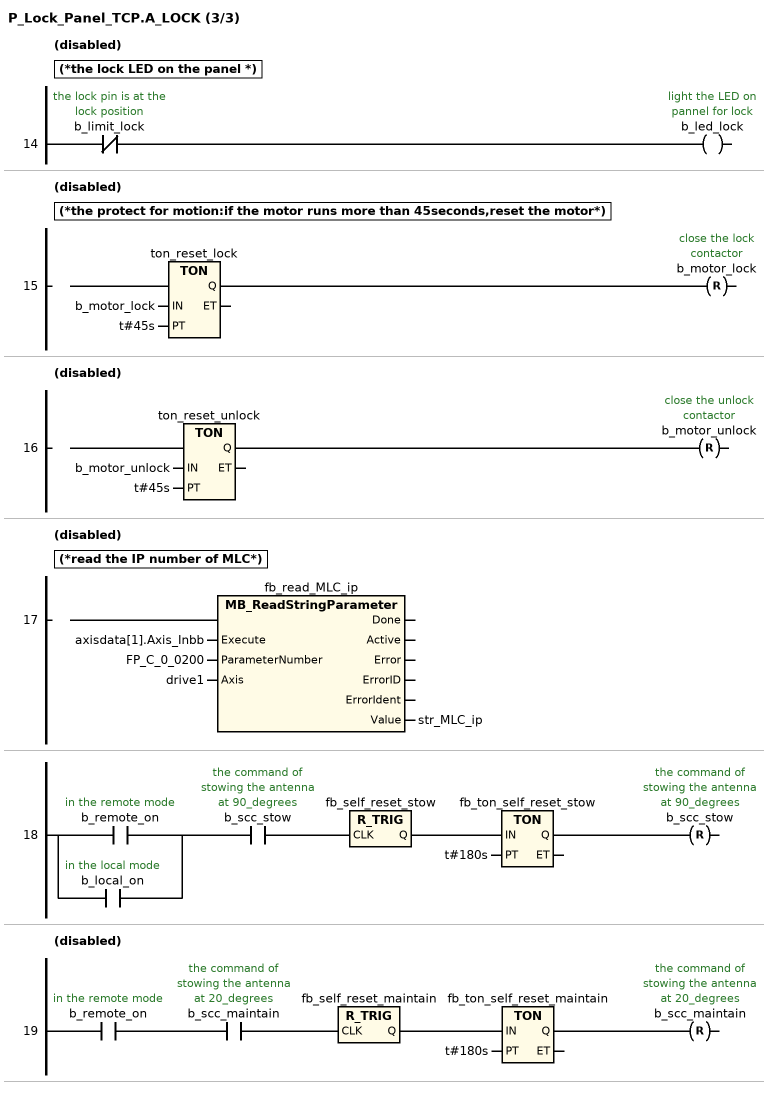
// NETWORK 14 (disabled)
//   b_limit_lock: the lock pin is at the lock position
//   b_led_lock: light the LED on pannel for lock
// label: (*the lock LED on the panel *)
// b_led_lock := NOT b_limit_lock;

// NETWORK 15 (disabled)
//   b_motor_lock: close the lock contactor
// label: (*the protect for motion:if the motor runs more than 45seconds,reset the motor*)
// ton_reset_lock(IN := b_motor_lock, PT := t#45s); // TON
// b_motor_lock R= ton_reset_lock.Q;

// NETWORK 16 (disabled)
//   b_motor_unlock: close the unlock contactor
// ton_reset_unlock(IN := b_motor_unlock, PT := t#45s); // TON
// b_motor_unlock R= ton_reset_unlock.Q;

// NETWORK 17 (disabled)
//   axisdata[1].Axis_Inbb: A-0-0021.13 -RD- Axis is ready for power to the amplifier (bb)
//   FP_C_0_0200: Engineering, IP address
//   drive1: Real axis "Drive1" with axis number 1
//   str_MLC_ip: IP number in MLC
// label: (*read the IP number of MLC*)
// fb_read_MLC_ip(
//     Execute := axisdata[1].Axis_Inbb,
//     ParameterNumber := FP_C_0_0200,
//     Axis := drive1,
//     Value => str_MLC_ip); // MB_ReadStringParameter

// NETWORK 18
//   b_remote_on: in the remote mode
//   b_local_on: in the local mode
//   b_scc_stow: the command of stowing the antenna at 90_degrees
fb_self_reset_stow(CLK := (b_remote_on OR b_local_on) AND b_scc_stow); // R_TRIG
fb_ton_self_reset_stow(IN := fb_self_reset_stow.Q, PT := t#180s); // TON
b_scc_stow R= fb_ton_self_reset_stow.Q;

// NETWORK 19 (disabled)
//   b_remote_on: in the remote mode
//   b_scc_maintain: the command of stowing the antenna at 20_degrees
// fb_self_reset_maintain(CLK := b_remote_on AND b_scc_maintain); // R_TRIG
// fb_ton_self_reset_maintain(IN := fb_self_reset_maintain.Q, PT := t#180s); // TON
// b_scc_maintain R= fb_ton_self_reset_maintain.Q;
END_ACTION

END_PROGRAM

// IndraMotionMlc1/Application/POUs/Panel Function/P_Panel_Jog
PROGRAM P_Panel_Jog
VAR
(*<<<<<<<<<<<<<<<azimuth>>>>>>>>>>>>>>>>*)
	r_vel_az: REAL;
	fb_panel_vel_az: MC_MoveVelocity;
	fb_panel_stop_az: MC_Stop;
	rtrig_panel_stop_az: R_TRIG;
	fb_blink_az: BLINK;
(*<<<<<<<<<<<<<<<elevation>>>>>>>>>>>>>>>*)
	r_vel_el: REAL;
	fb_panel_vel_el: MC_MoveVelocity;
	fb_panel_stop_el: MC_Stop;
	rtrig_panel_stop_el: R_TRIG;
	fb_blink_el: BLINK;
(*<<<<<<<<<<<<<FeedIndexer>>>>>>>>>>>>>>>>>*)
	r_vel_FI: REAL;
	fb_panel_vel_FI: MC_MoveVelocity;
	fb_panel_stop_FI: MC_Stop;
	rtrig_panel_stop_FI: R_TRIG;
	fb_blink_FI: BLINK;
(*the moving fuction into P_panel_jog program for FAT test and SAT test *)
	fb_test_move_az: MC_MoveAbsolute;
	fb_test_move_el: MC_MoveAbsolute;
	fb_test_move_FI: MC_MoveAbsolute;
	b_test_az: BOOL;
	b_test_el: BOOL;
	b_test_FI: BOOL;
	r_test_az: REAL;
	r_test_el: REAL;
	r_test_FI: REAL;
	r_test_vel_az:REAL;
	r_test_vel_el:REAL;
	r_test_vel_FI:REAL;
	b_test_az_r: BOOL;
	r_test_az_r: REAL;
	fb_test_relative_az: MC_MoveRelative;
	fb_test_relative_FI: MC_MoveRelative;
	r_test_FI_r: REAL;
	b_test_FI_r: BOOL;
END_VAR

(*<<<<<<<<<<<<<<<<<<<<<<<<<add the limit of the panel control>>>>>>>>>>>>>>>>>>>>>>>>*)
IF r_pos_az >= 358.5 THEN
	b_clockwise_AZ:= FALSE;
END_IF
IF r_pos_az <= -178.5 THEN
	b_cclockwise_AZ:= FALSE;
END_IF
IF r_pos_el >=90.1 THEN
	b_up_el:= FALSE;
END_IF
IF r_pos_el <=15 THEN
	b_down_el:=FALSE;
END_IF
IF r_pos_FI >= 178.5 THEN
	b_clockwise_FI:= FALSE;
END_IF
IF r_pos_FI <= -178.5 THEN
	b_cclockwise_FI:= FALSE;
END_IF

(*<<<<<<<<<<<<<<<<<<<<<<<set the azimuth speed value>>>>>>>>>>>>>>>>>>>>>>>>>>*)
IF b_clockwise_AZ = TRUE THEN
	IF b_speed_az = TRUE THEN
		r_vel_az:=0.5;
	ELSE
		r_vel_az:=0.17;
	END_IF
	IF r_pos_az>355 THEN
		r_vel_az:=0.17;
	END_IF
END_IF
IF b_cclockwise_AZ = TRUE THEN
	IF b_speed_az = TRUE THEN
		r_vel_az:=-0.5;
	ELSE
		r_vel_az:=-0.17;
	END_IF
	IF r_pos_az<-175 THEN
		r_vel_az:=-0.17;
	END_IF
END_IF
(*<<<<<<<<<<<<<<<<<<<<<<<set the elevation speed value>>>>>>>>>>>>>>>>>>>>>>>>>>*)
IF b_up_el =TRUE THEN
	IF b_speed_el = TRUE THEN
		r_vel_el:=0.17;
	ELSE
		r_vel_el:=0.05;
	END_IF
	IF r_pos_el>89 THEN
		r_vel_el:=0.05;
	END_IF
END_IF
IF b_down_el =TRUE THEN
	IF b_speed_el = TRUE THEN
		r_vel_el:=-0.17;
	ELSE
		r_vel_el:=-0.05;
	END_IF
	IF r_pos_el<16 THEN
		r_vel_el:=-0.05;
	END_IF
END_IF
(*<<<<<<<<<<<<<<<<<<<<<<<set the FeedIndexer speed value>>>>>>>>>>>>>>>>>>>>>>>>>>*)
IF b_clockwise_FI = TRUE THEN
	IF b_speed_FI = TRUE THEN
		r_vel_FI:=0.5;
	ELSE
		r_vel_FI:=0.17;
	END_IF
	IF r_pos_FI>175 THEN
		r_vel_FI:=0.17;
	END_IF
END_IF
IF b_cclockwise_FI = TRUE THEN
	IF b_speed_FI = TRUE THEN
		r_vel_FI:=-0.5;
	ELSE
		r_vel_FI:=-0.17;
	END_IF
	IF r_pos_FI<-175 THEN
		r_vel_FI:=-0.17;
	END_IF
END_IF

P_Panel_Jog.A_axes_running;

ACTION A_axes_running:
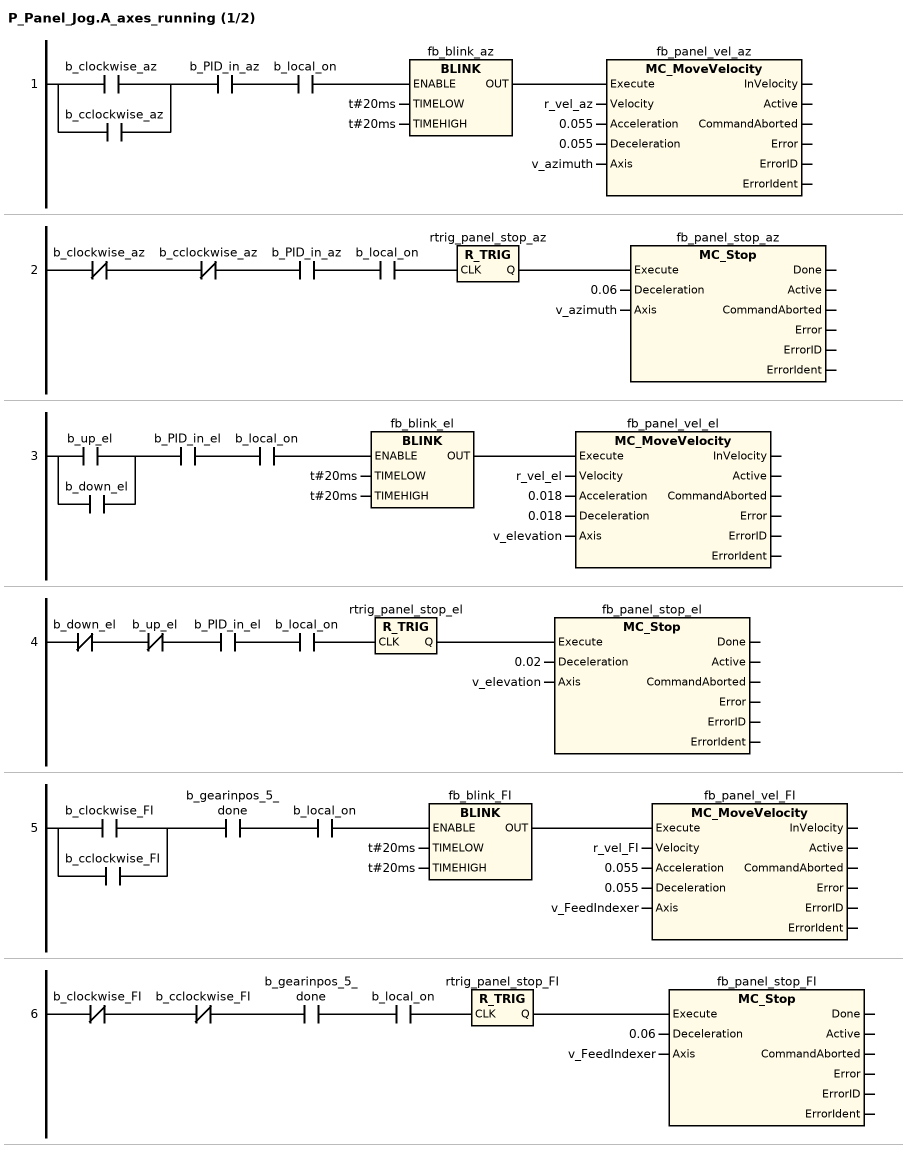
// NETWORK 1
fb_blink_az(
    ENABLE := (b_clockwise_az OR b_cclockwise_az) AND b_PID_in_az AND b_local_on,
    TIMELOW := t#20ms,
    TIMEHIGH := t#20ms); // BLINK
fb_panel_vel_az(
    Execute := fb_blink_az.OUT,
    Velocity := r_vel_az,
    Acceleration := 0.055,
    Deceleration := 0.055,
    Axis := v_azimuth); // MC_MoveVelocity

// NETWORK 2
rtrig_panel_stop_az(CLK := NOT b_clockwise_az AND NOT b_cclockwise_az AND b_PID_in_az AND b_local_on); // R_TRIG
fb_panel_stop_az(Execute := rtrig_panel_stop_az.Q, Deceleration := 0.06, Axis := v_azimuth); // MC_Stop

// NETWORK 3
fb_blink_el(
    ENABLE := (b_up_el OR b_down_el) AND b_PID_in_el AND b_local_on,
    TIMELOW := t#20ms,
    TIMEHIGH := t#20ms); // BLINK
fb_panel_vel_el(
    Execute := fb_blink_el.OUT,
    Velocity := r_vel_el,
    Acceleration := 0.018,
    Deceleration := 0.018,
    Axis := v_elevation); // MC_MoveVelocity

// NETWORK 4
rtrig_panel_stop_el(CLK := NOT b_down_el AND NOT b_up_el AND b_PID_in_el AND b_local_on); // R_TRIG
fb_panel_stop_el(Execute := rtrig_panel_stop_el.Q, Deceleration := 0.02, Axis := v_elevation); // MC_Stop

// NETWORK 5
fb_blink_FI(
    ENABLE := (b_clockwise_FI OR b_cclockwise_FI) AND b_gearinpos_5_done AND b_local_on,
    TIMELOW := t#20ms,
    TIMEHIGH := t#20ms); // BLINK
fb_panel_vel_FI(
    Execute := fb_blink_FI.OUT,
    Velocity := r_vel_FI,
    Acceleration := 0.055,
    Deceleration := 0.055,
    Axis := v_FeedIndexer); // MC_MoveVelocity

// NETWORK 6
rtrig_panel_stop_FI(CLK := NOT b_clockwise_FI AND NOT b_cclockwise_FI AND b_gearinpos_5_done AND b_local_on); // R_TRIG
fb_panel_stop_FI(Execute := rtrig_panel_stop_FI.Q, Deceleration := 0.06, Axis := v_FeedIndexer); // MC_Stop

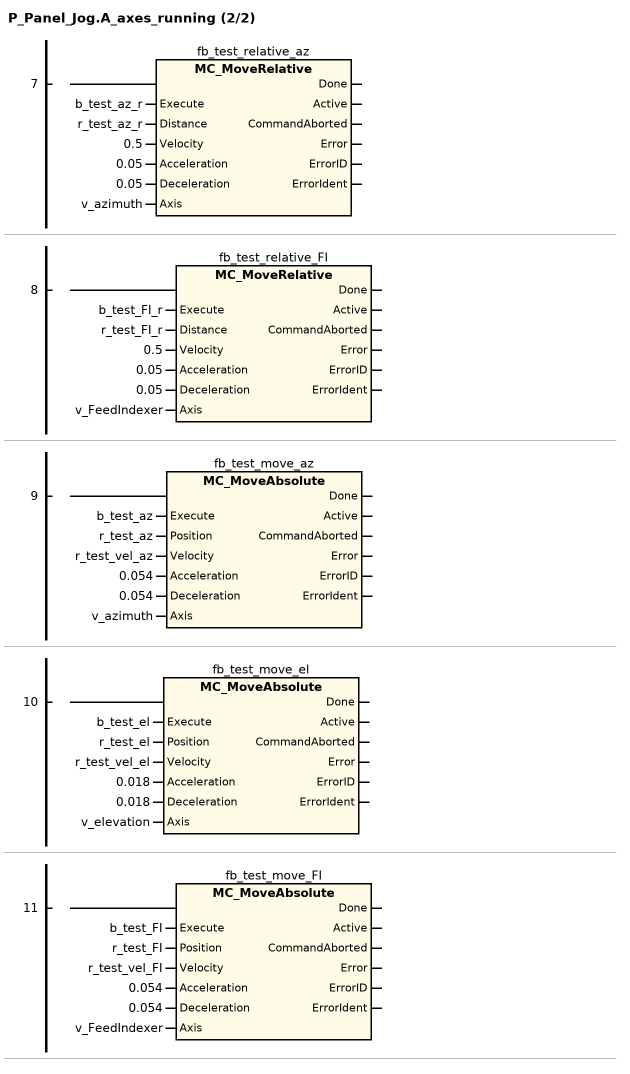
// NETWORK 7
fb_test_relative_az(
    Execute := b_test_az_r,
    Distance := r_test_az_r,
    Velocity := 0.5,
    Acceleration := 0.05,
    Deceleration := 0.05,
    Axis := v_azimuth); // MC_MoveRelative

// NETWORK 8
fb_test_relative_FI(
    Execute := b_test_FI_r,
    Distance := r_test_FI_r,
    Velocity := 0.5,
    Acceleration := 0.05,
    Deceleration := 0.05,
    Axis := v_FeedIndexer); // MC_MoveRelative

// NETWORK 9
fb_test_move_az(
    Execute := b_test_az,
    Position := r_test_az,
    Velocity := r_test_vel_az,
    Acceleration := 0.054,
    Deceleration := 0.054,
    Axis := v_azimuth); // MC_MoveAbsolute

// NETWORK 10
fb_test_move_el(
    Execute := b_test_el,
    Position := r_test_el,
    Velocity := r_test_vel_el,
    Acceleration := 0.018,
    Deceleration := 0.018,
    Axis := v_elevation); // MC_MoveAbsolute

// NETWORK 11
fb_test_move_FI(
    Execute := b_test_FI,
    Position := r_test_FI,
    Velocity := r_test_vel_FI,
    Acceleration := 0.054,
    Deceleration := 0.054,
    Axis := v_FeedIndexer); // MC_MoveAbsolute
END_ACTION

END_PROGRAM

// IndraMotionMlc1/Application/POUs/TCP/Message/FB_add_vector_old_mode
(* the function block is programmed for adding points to trajectory stack.
The input variables is type of string,and the output vaiable is the reply for TCP*)
FUNCTION_BLOCK FB_add_vector_old_mode
VAR_INPUT
	str_MJD:STRING;
	str_Azimuth:STRING;
	str_Elevation:STRING;
	str_FeedIndexer:STRING;
END_VAR
VAR_OUTPUT
	key:STRING;
END_VAR
VAR
(*(<<<<<<<<<<the transition variables>>>>>>>>>>>>>*)
	lreal_MJD: LREAL;
	real_azimuth: LREAL;
	real_elevation: LREAL;
	real_FeedIndexer: LREAL;
	tempAz:LREAL;
	tempEl:LREAL;
	temp_sin_Ao_C4:LREAL;
	temp_cos_Ao_C4:LREAL;
	temp_tanEo: LREAL;
	temp_sinE0:LREAL;
	temp_cosE0:LREAL;
	temp1:LREAL;
	temp2:LREAL;
	temp_R_sin_Ao_C4:LREAL;
	temp_R_cos_Ao_C4:LREAL;
	temp_R_tanEo:LREAL;
	temp_R_cosE0:LREAL;
	temp_R_sinE0:LREAL;
	temp1_exp:LREAL;
	temp2_exp:LREAL;
	new_Az:LREAL;
	new_El:LREAL;
	k:DINT;
	deltaAZ:LREAL:=0.0;
	deltaEL:LREAL:=0.0;
	aaaa:LREAL;
	bbbb:LREAL;
	test_1: LREAL;
END_VAR

(*lreal_MJD:=STRING_TO_LREAL(str_MJD)-0.000000076;*)(*set the ahead time for 6.6ms,so that the following error will be 0*)
lreal_MJD:=STRING_TO_LREAL(str_MJD);(*after gunner change P41 into 100ms,so the aheed time must be added by 50ms.(56.5ms)*)
real_azimuth:=STRING_TO_REAL(str_Azimuth);
real_Elevation:=STRING_TO_REAL(str_Elevation);
real_FeedIndexer:=STRING_TO_REAL(str_FeedIndexer);
deltaAZ:=0.0;
deltaEL:=0.0;
	tempAz:=real_azimuth;
    tempEl:=real_Elevation;
  		FOR k:=1 TO 3 BY 1 DO
        temp_sin_Ao_C4:=SIN(deg2rad(tempAz-C4));
        temp_cos_Ao_C4:=COS(deg2rad(tempAz-C4));
        temp_tanEo:=TAN(deg2rad(tempEl));
        temp_cosE0:=COS(deg2rad(tempEl));
        temp_sinE0:=SIN(deg2rad(tempEl));
        temp1:=tempAz-(C1+C3*temp_sin_Ao_C4*temp_tanEo+C5*temp_tanEo+C6/temp_cosE0);
        temp2:=tempEl-(C2+C3*temp_cos_Ao_C4+C7*temp_cosE0);
        temp_R_sin_Ao_C4:=SIN(deg2rad(temp1-C4));
        temp_R_cos_Ao_C4:=COS(deg2rad(temp1-C4));
        temp_R_tanEo:=TAN(deg2rad(temp2));
        temp_R_cosE0:=COS(deg2rad(temp2));
        temp_R_sinE0:=SIN(deg2rad(temp2));
        temp1_exp:=temp1+C1+C3*temp_R_sin_Ao_C4*temp_R_tanEo+C5*temp_R_tanEo+C6/temp_R_cosE0;
        temp2_exp:=temp2+C2+C3*temp_R_cos_Ao_C4+C7*temp_R_cosE0;
        deltaAz:=real_azimuth-temp1_exp;
        deltaEl:=real_Elevation-temp2_exp;
        tempAz:=tempAz+deltaAz;
        tempEl:=tempEl+deltaEl;
    END_FOR;
	new_Az:=temp1;
	new_El:=Encoder_to_motor(temp2);
	aaaa:=new_Az-real_azimuth;
	bbbb:=new_El-real_Elevation;
(*<<<<<<<<<<<<<<<<<<<<<<<<<<<<<<<judgement according to ICD document>>>>>>>>>>>>>>>>>>>>>>>>>>>>>>>*)

test_1:=lreal_MJD-lr_MJD_current;
IF (lreal_MJD-lr_MJD_current)>0.001 THEN	
IF real_azimuth>=-270 AND real_azimuth<=270 AND real_elevation>=15 AND real_elevation<=90 AND real_FeedIndexer>=0 AND real_FeedIndexer<=180 THEN
	IF lreal_MJD> (track_table[i_End].MJD) THEN
		IF i_num_stack_left<i_total THEN
			IF track_table[i_end].MJD<>0 THEN
				i_end:=F_I_number(i_end+1);
			END_IF;
			key:='OK';
			track_table[i_End].MJD:=lreal_MJD;
			track_table[i_End].Azimuth:= new_Az;//-0.2884;
			track_table[i_End].Elevation:= new_El;
			track_table[i_End].FeedIndexer:= tempEl;
			track_table[i_End].Elevation_ori:=temp2;
		ELSE
			key:='NAK - Stack is full';
		END_IF;
	ELSE
		key:='NAK - MJD is out of sequence';
	END_IF;
ELSE
	key:='NAK - One or more trkval coords are unreachable';
END_IF;
END_IF;

END_FUNCTION_BLOCK

// IndraMotionMlc1/Application/POUs/TCP/Message/FB_MSG
(*This program is built for find the key word and transfer sub-program to
distill the keyword from the message*)
FUNCTION_BLOCK FB_MSG
VAR_INPUT
	str_Message:STRING;
END_VAR
VAR_OUTPUT
	Key:STRING;
	P_value: ARRAY [1..10] OF STRING;
END_VAR
VAR
	MSG_Divide : FB_Str_Divide;(*transfer  the function block *)
	Head:STRING:='to_MLC';(*defination of recieved head*)
	Str_MSG: STRING;(*transition value*)
	int_MSG: INT;
	int_Len: USINT;
	str_Head: STRING;
	Counter: INT;
END_VAR

(*clear key and P_value*)
key:='';
FOR Counter:=1 TO 10 BY 1 DO
	P_value[counter]:='';
END_FOR;
Str_MSG:=str_Message;
str_head:=LEFT(Str_MSG,6);(*read the received head*)
str_MSG:=RIGHT(str_msg,LEN(str_msg)-6);
(*judge the head of the message whether is to_MLC,if it is true, transfer sub-program
to distill the keyword1,keyword2,keyword3 and so on*)
IF str_head<>head THEN
	Key:='NAK Head Error';
ELSE
	int_Len:=STRING_TO_USINT(LEFT(str_msg,4));
	str_MSG:=RIGHT(str_msg,LEN(str_msg)-4);

	MSG_Divide(input_str:=Str_MSG);
	key:=MSG_Divide.Output_str1;
	Str_MSG:=MSG_Divide.Output_str2;
(*enable*)
 	IF key ='ENABLE' THEN
		MSG_Divide(input_str:=Str_MSG);
		P_value[1]:=MSG_Divide.Output_Str1;
(*estop*)
	ELSIF	key ='ESTOP' THEN
		P_value[1]:='';
(*goto*)
	ELSIF	key ='GOTO' THEN
		MSG_Divide(input_str:=Str_MSG);
		P_value[1]:=MSG_Divide.Output_Str1;
		Str_MSG:=MSG_Divide.Output_str2;
		MSG_Divide(input_str:=Str_MSG);
		P_value[2]:=MSG_Divide.Output_Str1;
		Str_MSG:=MSG_Divide.Output_str2;
		MSG_Divide(input_str:=Str_MSG);
		P_value[3]:=MSG_Divide.Output_Str1;
(*setmovevelocity*)
	ELSIF	key ='SETSPEED' THEN
		MSG_Divide(input_str:=Str_MSG);
		P_value[1]:=MSG_Divide.Output_Str1;
		Str_MSG:=MSG_Divide.Output_str2;
		MSG_Divide(input_str:=Str_MSG);
		P_value[2]:=MSG_Divide.Output_Str1;
		Str_MSG:=MSG_Divide.Output_str2;
		MSG_Divide(input_str:=Str_MSG);
		P_value[3]:=MSG_Divide.Output_Str1;	
(*velpos*)
    ELSIF	key ='VELPOS' THEN
		MSG_Divide(input_str:=Str_MSG);
		P_value[1]:=MSG_Divide.Output_Str1;
		
		Str_MSG:=MSG_Divide.Output_str2;
		MSG_Divide(input_str:=Str_MSG);
		P_value[2]:=MSG_Divide.Output_Str1;
		
		Str_MSG:=MSG_Divide.Output_str2;
		MSG_Divide(input_str:=Str_MSG);
		P_value[3]:=MSG_Divide.Output_Str1;
		
		Str_MSG:=MSG_Divide.Output_str2;
        MSG_Divide(input_str:=Str_MSG);
		P_value[4]:=MSG_Divide.Output_Str1;
		
		Str_MSG:=MSG_Divide.Output_str2;
		MSG_Divide(input_str:=Str_MSG);
		P_value[5]:=MSG_Divide.Output_Str1;
		
		Str_MSG:=MSG_Divide.Output_str2;
		MSG_Divide(input_str:=Str_MSG);
		P_value[6]:=MSG_Divide.Output_Str1;	        	
	
(*GSTAT*)
	ELSIF	key ='GSTAT' THEN
		P_value[1]:='';
(*UPDATE*)
	ELSIF	key ='UPDATE' THEN
		P_value[1]:='';
(*KSTAT*)
	ELSIF	key ='K1STAT' THEN
		P_value[1]:='';
	ELSIF	key ='K2STAT' THEN
		P_value[1]:='';
	ELSIF	key ='K3STAT' THEN
		P_value[1]:='';
	ELSIF	key ='K4STAT' THEN
		P_value[1]:='';
	ELSIF	key ='K5STAT' THEN
		P_value[1]:='';
	ELSIF	key ='VERSION' THEN
		P_value[1]:='';
(*PWR*)
	ELSIF	key ='PWR' THEN
		MSG_Divide(input_str:=Str_MSG);
		P_value[1]:=MSG_Divide.Output_Str1;
(*STOP*)
	ELSIF	key ='STOP' THEN
		P_value[1]:='';
(*STOW*)
	ELSIF	key ='HOME' THEN
		P_value[1]:='';
(*STOW*)
	ELSIF	key ='STOW' THEN
		P_value[1]:='';
(*MAINTAIN*)
	ELSIF	key ='MAINTAIN' THEN
		P_value[1]:='';
(*UNLOCK*)
	ELSIF	key ='UNLOCK' THEN
		P_value[1]:='';
(*UNLOCK*)
	ELSIF	key ='LOCK' THEN
		P_value[1]:='';
(*TRACK*)
	ELSIF	key ='TRACK' THEN
		MSG_Divide(input_str:=Str_MSG);
		P_value[1]:=MSG_Divide.Output_Str1;
(*TRKVAL*)
	ELSIF	key ='TRKVAL' THEN
			MSG_Divide(input_str:=Str_MSG);
			P_value[1]:=MSG_Divide.Output_Str1;
			Str_MSG:=MSG_Divide.Output_str2;
			MSG_Divide(input_str:=Str_MSG);
			P_value[2]:=MSG_Divide.Output_Str1;
			Str_MSG:=MSG_Divide.Output_str2;
			MSG_Divide(input_str:=Str_MSG);
			P_value[3]:=MSG_Divide.Output_Str1;
			Str_MSG:=MSG_Divide.Output_str2;
			MSG_Divide(input_str:=Str_MSG);
			P_value[4]:=MSG_Divide.Output_Str1;
			
(*VEL*)
	ELSIF	key ='VEL' THEN
			MSG_Divide(input_str:=Str_MSG);
			P_value[1]:=MSG_Divide.Output_Str1;
			Str_MSG:=MSG_Divide.Output_str2;
			MSG_Divide(input_str:=Str_MSG);
			P_value[2]:=MSG_Divide.Output_Str1;
			Str_MSG:=MSG_Divide.Output_str2;
			MSG_Divide(input_str:=Str_MSG);
			P_value[3]:=MSG_Divide.Output_Str1;
(*UPDATE*)
	ELSIF	key ='SNTP' THEN
		P_value[1]:='';	
(*LOCKSTANDBY*)
	ELSIF	key ='LOCKSTANDBY' THEN
		P_value[1]:='';		
(*OFFSET*)
	ELSIF	key ='OFFSET' THEN
		MSG_Divide(input_str:=Str_MSG);
		P_value[1]:=MSG_Divide.Output_Str1;
		Str_MSG:=MSG_Divide.Output_str2;
		MSG_Divide(input_str:=Str_MSG);
		P_value[2]:=MSG_Divide.Output_Str1;						
(*TSTAT*)
	ELSIF	key ='TSTAT' THEN
		P_value[1]:='';
(*<<<<<<<<<<<<<<<<<<<<<<other>>>>>>>>>>>>>>>>>>>>>>>>>>>>*)
	ELSE
		key:='NAK Key Error';
	END_IF;
END_IF;

END_FUNCTION_BLOCK

// IndraMotionMlc1/Application/POUs/TCP/Message/FB_Str_Divide
(*This program is built for divide the headword and keyword
from the receive message,the theory is divide the words by every 'space'*)
FUNCTION_BLOCK FB_Str_Divide
VAR_INPUT
	Input_str:STRING;
END_VAR
VAR_OUTPUT
	Output_str1:STRING;
	Output_Str2:STRING;
END_VAR
VAR
	Str_MSG: STRING;
	int_MSG: INT;
	int_Len: UINT;
END_VAR

(*transfer the sub-program F_Trim to trim message,then find the 'space'*)
input_str:=F_Trim(input_str);
int_MSG := FIND (Input_str ,' ');
int_Len:=LEN (Input_str);
(*if there is no words behind the 'spcae',end the process of dividing message*)
IF int_MSG=0 THEN
Output_str1:=Input_str;
ELSE
(*if there is still some words behind the 'space',continue the process of dividing message*)
Output_str1:=LEFT(Input_str,int_MSG-1);
Output_str2:=F_Trim(RIGHT(Input_str,int_len-int_MSG));
END_IF

END_FUNCTION_BLOCK

// IndraMotionMlc1/Application/POUs/TCP/Message/F_Trim
(*This program is built for distilling the key from the message that had received*)
FUNCTION F_Trim : STRING(255)
VAR_INPUT
	Str_intput:STRING(255);
END_VAR
VAR
	Counter: UINT;
	Uint_len: UINT;
END_VAR

WHILE LEFT(Str_intput,1)=' ' DO
	Uint_len:=LEN(Str_intput);
	Str_intput:=RIGHT(Str_intput,Uint_len-1);
END_WHILE
F_Trim:=Str_intput;

END_FUNCTION

// IndraMotionMlc1/Application/POUs/TCP/Message/F_RPL
(*This program is bulit for combining the head string and message string together,and calculate
the amount of the whole string,the final string will be sent by TCP*)
FUNCTION F_RPL : STRING(1500)
VAR_INPUT
		key:STRING(1500);
	message:STRING(1500);
END_VAR
VAR
	str_Head:STRING:='fr_MLC';
	str_text:STRING(1500);
	str_text2: STRING(1500);
	int_len_head: INT;
END_VAR

(*If the massage is not null, then evaluate the str_text*)
IF message<>'' THEN
	str_text:=CONCAT(' - ',message);
END_IF;
(*combining the key string and message string*)
str_text:=CONCAT(key,str_text);
(*calculate the amount of the str_text*)
int_len_head:=LEN(str_text);
(*According to the amount of the str_text,add appropriate space to fit 4bits*)
IF int_len_head<10 THEN
	str_text2:=CONCAT('   ',INT_TO_STRING(int_len_head));
ELSIF int_len_head<100 AND int_len_head>=10 THEN
	str_text2:=CONCAT('  ',INT_TO_STRING(int_len_head));
ELSIF int_len_head<1000 AND int_len_head>=100 THEN
	str_text2:=CONCAT(' ',INT_TO_STRING(int_len_head));
ELSE
	str_text2:=INT_TO_STRING(int_len_head);
END_IF
(*combining all the need strings and calculate the length*)
str_text:=CONCAT(str_text2,str_text);
F_RPL:=CONCAT(str_Head,str_text);
ui_Length_Reply:=LEN(F_RPL);

END_FUNCTION

// IndraMotionMlc1/Application/POUs/TCP/Message/F_RPL_1
(*This program is bulit for combining the head string and message string together,and calculate
the amount of the whole string,the final string will be sent by TCP*)
FUNCTION F_RPL_1 : STRING(1000)
VAR_INPUT
		key:STRING(1000);
	message:STRING(1000);
END_VAR
VAR
	str_Head:STRING:='fr_MLC';
	str_text:STRING(1000);
	str_text2: STRING(1000);
	int_len_head: INT;
END_VAR

(*If the massage is not null, then evaluate the str_text*)
IF message<>'' THEN
	str_text:=CONCAT(' - ',message);
END_IF;
(*combining the key string and message string*)
str_text:=CONCAT(key,str_text);
(*calculate the amount of the str_text*)
int_len_head:=LEN(str_text);
(*According to the amount of the str_text,add appropriate space to fit 4bits*)
IF int_len_head<10 THEN
	str_text2:=CONCAT('   ',INT_TO_STRING(int_len_head));
ELSIF int_len_head<100 AND int_len_head>=10 THEN
	str_text2:=CONCAT('  ',INT_TO_STRING(int_len_head));
ELSIF int_len_head<1000 AND int_len_head>=100 THEN
	str_text2:=CONCAT(' ',INT_TO_STRING(int_len_head));
ELSE
	str_text2:=INT_TO_STRING(int_len_head);
END_IF
(*combining all the need strings and calculate the length*)
str_text:=CONCAT(str_text2,str_text);
F_RPL_1:=CONCAT(str_Head,str_text);
ui_Length_Reply:=LEN(F_RPL_1);

END_FUNCTION

// IndraMotionMlc1/Application/POUs/TCP/Message/F_RPL_2
(*This program is bulit for combining the head string and message string together,and calculate
the amount of the whole string,the final string will be sent by TCP*)
FUNCTION F_RPL_2 : STRING(1500)
VAR_INPUT
		key:STRING(1500);
	message:STRING(1500);
END_VAR
VAR
	str_Head_F:STRING:='F';
	str_text:STRING(1500);
	str_text2: STRING(1500);
	int_len_head: INT;
END_VAR

(*If the massage is not null, then evaluate the str_text*)
IF message<>'' THEN
	str_text:=CONCAT(' - ',message);
END_IF;
(*combining the key string and message string*)
str_text:=CONCAT(key,str_text);
(*calculate the amount of the str_text*)
int_len_head:=LEN(str_text);
(*According to the amount of the str_text,add appropriate space to fit 4bits*)
IF int_len_head<10 THEN
	str_text2:=CONCAT('   ',INT_TO_STRING(int_len_head));
ELSIF int_len_head<100 AND int_len_head>=10 THEN
	str_text2:=CONCAT('  ',INT_TO_STRING(int_len_head));
ELSIF int_len_head<1000 AND int_len_head>=100 THEN
	str_text2:=CONCAT(' ',INT_TO_STRING(int_len_head));
ELSE
	str_text2:=INT_TO_STRING(int_len_head);
END_IF
(*combining all the need strings and calculate the length*)
str_text:=CONCAT(str_text2,str_text);
F_RPL_2:=CONCAT(str_Head_F,str_text);
ui_Length_Reply:=LEN(F_RPL_2);

END_FUNCTION

// IndraMotionMlc1/Application/POUs/Annotation
PROGRAM Annotation
VAR
	Annotation_version : REAL;
END_VAR

Annotation_version:=1.01;
(*
                               The Annotation of Program

	This program is built for controlling the ASKAP antennas in Australia. It based on the
Indrologic software and been embedded in the MLC. 

	The program is made up of four parts:

	Firstly, the program in the folder named 'Motion'include some basal operation that can 
be used by panelbox(local) and TCP command(remote). In this section we can give the power 
and enable to each axis,tansfer the function block for antibacklash and set the value of limit.
And,the P_Track program run the antenna to follow the trajectory.

	Secondly, the Panel Function is built for realizing the manual operating.it involves controlling
the antenna to move,reading the drive I/O,lighten the led and switching the local mode or remote mode.
All of these are operated on the panelbox.

	Thirdly, the TCP is bulit for remote controlling. It involves receiving the message from CSIRO, analysing
and disposing the command, carrying out the action and sending the message to CSIRO.

	Fourthly, the Time Control folder write for updata the system time in order to insuring the 
correctness of trajectory.



								History of Version
Version 1.02(2014-8-27)
	Hardware:     1.None 
	Improvement:  1. change the bias to 0 when the drive enable off.
				  2. change the strategy of the first trajectory point.


Version 1.02(2014-7-16)
	Hardware:     1.None 
	Improvement:  1. reset some variables that effect on the goto and stow function by received the command 'POWER OFF' and 'ENABLE OFF'. 

Version 1.01(2013-4-19)
	Hardware:     1.None 
	Improvement:  1. change the judgment about the zero velocity

Version 1.0(2012-10-19)
	Hardware:     1.None 
	Improvement:  1. Change the final program version number to 1.0.

Version 0.86(2012-09-19)
	Hardware:     1.None 
	Improvement:  1. retain the list of the PID parameters but make the list noneffective .

Version 0.85(2012-08-12)
	Hardware:     1.None 
	Improvement:  1. add the list of the PID parameters .
 
Version 0.84(2012-05-28)
	Hardware:     1.None 
	Improvement:  1. add the motion limit in local mode .
				  2. change the action when track off 
				  3. fix the problem of power_on and power_off .

Version 0.83(2012-05-14)
	Hardware:     1.None 
	Improvement:  1. fix the problem of the GOTO function.
				  2. add the automatic adjustment of the azimuth axis PID parameters.
				  3. improve the method of the elevation power.

Version 0.82(2012-03-23)
	Hardware:     1.None 
	Improvement:  1. adjust the overtemp from 145 degree to 70 degree
				  2. add a new main status bit to show if the axis shutdown by overtemp or overcurrent
                  3. add a action to shutdown the axis when it overtemp or overcurrent 

Version 0.81(2011-10-26)
	Hardware:     1.adjust the EL limit to below 15 
	Improvement:  1. enlarge the window of driving or locked
                  2. add a new main status bit to show the status of lock motor
				  3. add a new axis status bit to show the track overspeed 
				  4. add a array to store the NTP server IP address
 
Version 0.8(2011-07-05)
	Hardware:     1.None.
	Improvement:  1. add a delay to control the b_SCC_STOW self resetting
                  2. improve the program so that the stow action can be canceled during the process of moving the EL to 90

Version 0.7(2011-06-20)
	Hardware:     1.None.
	Improvement:  1. change the method of power on,so that the EL can re-enable in the softlimit position

Version 0.6(2011-06-06)
	Hardware:     1.The parameters of the servo loop is refined  FeedIndexer.
	Improvement:  1.change the P_panel_jog program for preventing the wrong direction.
				  2.delete the 1sec delay in P_power_on_TCP.
				  3.add the error message for the broken connection of the limit cables.

Version 0.5(2011-03-25)
	Hardware:     1.The parameters of the servo loop is refined by the Germen engineer.
				  2.Add a fan for MLC.			
	New function: 1.the moving fuction into P_panel_jog program for FAT test and SAT test 
				  2.the function of disabling all the axises when the connection is broken unwittingly.
				  3.add K4STAT command into P_TCP_with_SCC to check the system.
	Improvement:  1.change the trajectory mode from parabolic curve into cubic curve.
				  2.modify the blackbox fuction,IP number is 192.168.1.1xx and port is 4343.
				  3.modify the parameters of PID for antibacklash.
				  4.the fuction of showing the position values beyond the normal.
				  5.increase the operator pendant wrap warning limits.

Version 0.4(2010-10-28)

	Hardware:     1.MLC is L65.
				  2.The control section of drive is MPH05.

	New function: 1.judgement the stow position according to the IP number.
				  2.change the method of running trajectory.

	Improvement:  1.protection for the lock limit.
				  2.remove the ralative parameters form the stack.

Version 0.3(2010-8-8)

	Hardware:     1.MLC is changed from L40 to L65.
				  2.The control section of drive is advanced to MPH05.
	
	New function: 1.add the clicker fuction of the panel LED for the judgement of position.
				  2.add the enable switch for azimuth,elevation and FeedIndexer.
				  3.add the new command according to the new ICD.
				  4.add the panel estop status.

	Improvement:  1.the module of time master axis is changed from 3600 to 900.
				  2.use the new trajectory,X_MOTION_IN_MOTION_FIY5_SLIM.

Version 0.2(2010-04-05)

	Hardware:     1.MLC is L40.
				  2.The control section of drive is MPB04.	

	New function: 1.protection of loss power
				  2.protection of lock position
				  3.report the operation_hour
				  4.report the diagnosis of each drive

	Improvement:  1.improve the new arithmetic of NTP,it can solve the leapyear problem				 
				  2.other small problems for stability

Version 0.1(2009-10-01)

	Hardware:     1.MLC is L40.
				  2.The control section of drive is MPB04.	

	Basal function: 1.Power and enable
					2.panel control
					3.TCP communication
					4.NTP 
					5.track

When you are reading the program and you want to know more information,
you can call for the help,by pushing the F1 button after choosing the type. 
for example:
The function block R_TRIG detects a rising edge. 
The function block F_TRIG detects a falling edge
The function block TON implements a turn-on delay
A_xxxxxx means a sub-program.

Self-test of control system:(K4STAT)
You can send K4STAT command on TCP to check the control system 
if the reply involve the code of 'Exxxx' or 'Fxxxx'or 'Cxxxx',which canot be cleared,there is something wrong in control system.

*)

END_PROGRAM

// IndraMotionMlc1/Application/POUs/TCP/P_TCP_with_SCC
(*This program is built for TCP communication, receive the message from CSIRO,deal with the commands,and send the reply to CSIRO*)
PROGRAM P_TCP_with_SCC
VAR
(*<<<<<<<<<<<<<<<<<<<<<<<<<<<<<<<<<<<<<<<<<<<>>>>>>>>>>>>>>>>>>>>>>>>>>>>>>>>>>>>>*)
	b_receiving :BOOL;
	b_commanding: BOOL;
	b_sending: BOOL;
	str_MSG_Received:STRING(255);(*the received message*)
	fb_MSG_receive :FB_MSG;(*transfer the defined function block,FB_MSG*)
	fb_Trkval:FB_add_vector;(*transfer the defined function block,FB_add_vector*)
	b_Scc_PWR_on: BOOL;
	b_Scc_PWR_off: BOOL;
(*<<<<<<<<<<<<<<<<<<<<<<<<<<<<<<<<<<<<<<<<<<<CONNECTION>>>>>>>>>>>>>>>>>>>>>>>>>>>>>>>>>>>>>*)
	TCPConnection: IL_UDPSocketAsync;
	b_Server_Enable: BOOL:=TRUE;(*the enable of IL_TCPConnectionAsync*)
	di_Socket: DINT;(*the socket number*)
//	strIP: STRING;
	strIP: STRING:='192.168.1.111';
	b_Connection_done: BOOL;
(*<<<<<<<<<<<<<<<<<<<<<<<<<<<<<<<<<<<<<<<<<<<RECEIVE>>>>>>>>>>>>>>>>>>>>>>>>>>>>>>>>>>>>>*)
	TCPRecv:IL_UDPRecvfromAsync ;
	b_Recv_enable: BOOL;
	b_Recv_done: BOOL;
	str_Recv: STRING(255);
	di_ReceivedBytes: DINT;
(*<<<<<<<<<<<<<<<<<<<<<<<<<<<<<<<<<<<<<<<<<<<<SEND>>>>>>>>>>>>>>>>>>>>>>>>>>>>>>>>>>>>>*)
	TCPSend: IL_UDPSendtoAsync;
	b_Send_enable: BOOL;
	b_Send_done: BOOL;
	str_Send: STRING(1000);
	di_SentBytes: DINT;
(*<<<<<<<<<<<<<<<<<<<<<<<<<<<<<<<<<<<<<<<<<<<<<<<<<<<power>>>>>>>>>>>>>>>>>>>>>>>>>>>>>>>>>>>>*)
	ton_pow_off_az: TON;
	ton_pow_off_el: TON;
	ton_pow_off_FI: TON;
	rtrig_power_az: R_TRIG;
	rtrig_power_el: R_TRIG;
	rtrig_power_FI: R_TRIG;
	fb_ton_el: TON;
	fb_ton_FI: TON;
	rtrig_off_az: R_TRIG;
	rtrig_off_el: R_TRIG;
	rtrig_off_FI: R_TRIG;
	b_clear_err: BOOL;
	FB_clear_error_off: MB_WriteParameter;
	b_clear_off_done: BOOL;
	rtrig_err: R_TRIG;
	rtrig_clear_done: R_TRIG;
(*<<<<<<<<<<<<<<<<<<<<<<<<<<<<<<<<<<<<stop>>>>>>>>>>>>>>>>>>>>>>>>>>>>>*)
	b_stop1_done: BOOL;
	b_stop3_done: BOOL;
	b_stop5_done: BOOL;
	fb_scc_stop1: MC_Stop;
	fb_scc_stop3: MC_Stop;
	fb_scc_stop5: MC_Stop;
	rtrig_stop_az: R_TRIG;
	rtrig_stop_el: R_TRIG;
	rtrig_stop_FI: R_TRIG;
	b_stop_act_az: BOOL;
	b_stop_act_el: BOOL;
	b_stop_act_FI: BOOL;
	rtrig_reset_stop: R_TRIG;
(*<<<<<<<<<<<<<<<<<<<<<<<<<<<<<<<<<<<<<<<<<<<GOTO>>>>>>>>>>>>>>>>>>>>>>>>>>>>>>>>>>>>>>>>>>>*)


	fb_goto_Az: MC_MoveRelative;
	fb_goto_El: MC_MoveAbsolute;
	fb_goto_FI: MC_MoveRelative;
	b_active_AZ: BOOL;
	b_active_el: BOOL;
	b_active_FI: BOOL;
	rtrig_goto: R_TRIG;
(*K3STAT*)
	status_K3:DWORD;
(*add the function of close TCP function*)
	fb_tcp_close: IL_UDPCloseAsync;
	B_TCP_close: BOOL;
	b_TCP_close_done: BOOL;
	b_Recv_active: BOOL;
	i_counter_tcp:INT;
	rtrig_stop_stow: R_TRIG;
	Ftrig_goto: R_TRIG;
(*************vel**************)
r_vel_az:REAL;
r_vel_el:REAL;	
r_vel_FI:REAL;	

	
	rttig_vel: R_TRIG;
	b_scc_vel1: BOOL;
	fb_vel_az: MC_MoveVelocity;
	b_vel_az_done: BOOL;
	b_active_vel_az: BOOL;
	fb_vel_el: MC_MoveVelocity;
	b_active_vel_el: BOOL;
	b_vel_el_done: BOOL;
	fb_vel_FI: MC_MoveVelocity;
	b_active_vel_FI: BOOL;
	b_vel_FI_done: BOOL;
	fb_r_vel1: R_TRIG;
	fb_r_vel2: R_TRIG;
	fb_f_vel3: F_TRIG;
	fb_f_vel4: F_TRIG;
	fb_r_vel5: R_TRIG;
	fb_ton_vel: ton;
	str_concat: ARRAY[1..40] OF STRING(1000);(*数组及其类型的定义*)	
	Counter: INT;
	bWaiting4Connection: BOOL;
	bConnError: BOOL;
	diConnError: ERROR_CODE;
	ConnectError: ERROR_STRUCT;
i_counter_1s: INT:=0;	
	r_offset_az_I: REAL;
	r_offset_el_I: REAL;
	rtrig_power_power: R_TRIG;
	i_count:INT;
	
(*the status word for GSTAT*)	
	status_1:DWORD;
	status_2:DWORD;
	status_3:DWORD;
	status_4:DWORD;
	status_5:DWORD;
	status_6:DWORD;
(*the status code*)	
    drive_code1:STRING;
	drive_code2:STRING;
	drive_code3:STRING;
	drive_code4:STRING;
	drive_code5:STRING;
	drive_code6:STRING;

	
	vel_move_az: REAL:=0.3;
	vel_move_el: REAL:=0.167;
	vel_move_FI: REAL:=0.333;
	
	r_a0:REAL;
	v_a0:REAL;
	a_a0:REAL;
	t_difference:REAL;
	b_test:BOOL;
	
	r_az_pause_pos1:REAL;
	r_az_pause_pos2:REAL;
	r_az_pause_pos3:REAL;
	r_az_pause_pos4:REAL;
	r_az_pause_pos5:REAL;
	r_az_pause_pos6:REAL;
	r_az_pause_pos7:REAL;
	i_pause_temp:INT;
	
	fb_f_track_on:F_TRIG;
	b_not_track:BOOL;
	i_count_stop:INT;
	i_stop:INT;
	i_stop_1:INT;
	b_stop_TOA:BOOL;
	
	b_limit_az:BOOL;
	b_limit_el:BOOL;
	b_limit_FI:BOOL;
	
	fb_r_az_limit:r_trig;
	fb_r_el_limit:r_trig;
	fb_r_FI_limit:r_trig;
	
	i_new_cmd_dalay:DINT:=0;
	
	acc_mov_az: REAL;
	dcc_mov_az: REAL;
	vel_move_az_1: REAL;
	fb_start_goto_az: R_TRIG;
	b_moving: BOOL;
	fb_start_goto_az1: R_TRIG;
	fb_blink_move_az: BLINK;

	bTESTTTT: BOOL;
	fb_vel_el_1: MC_MoveVelocity;
	RTESTE: REAL;
	r_p1: LREAL;
	r_p0: LREAL;
	r_p2: LREAL;
	vel_stop_ton:TON;
	
	reply_count: DINT;
	TON_0: ton;
	FB_move_master_az1: MC_MoveAbsolute;
	b_Stop_Az: BOOL;
	b_start_goto_az_tcp: BOOL;
END_VAR


fb_f_track_on(clk:=b_track_on);

 IF b_goto_Az_done THEN
	b_step_running_az:=FALSE; 
 END_IF
 
 IF b_step_running_az=0 AND b_step_running_el=0 THEN
	 b_step_running:=0;
 END_IF
 IF b_step_running_az AND b_step_running_el THEN
	 b_step_running:=1;
 END_IF
 
 IF b_step_running OR b_offset_running THEN
	IF b_step_running THEN
	 r_step_count:=r_step_count_temp;
	END_IF 
	IF b_offset_running THEN
	 r_step_count:=r_offset_count_temp;
	END_IF 
 ELSE
	 r_step_count:=0;
 END_IF
	
 
 
 

	
IF fb_f_track_on.Q THEN
	b_not_track:=TRUE;	
END_IF

IF b_not_track AND i_num_stack_left=0 THEN
		i_start:=1;
		i_end:=1;
		track_table[1].TAIoffset:=0;
		FOR i_count:=1 TO i_total BY 1 DO
			track_table[i_count].TAIoffset:=0;
			track_table[i_count].Azimuth:= 0;
			track_table[i_count].Elevation:=0;
			//track_table[i_count].FeedIndexer:=0;
		END_FOR;
		(*track_table[1].MJD:=0;
		FOR i_count:=1 TO i_total BY 1 DO
			track_table[i_count].MJD:=0;
			track_table[i_count].Azimuth:= 0;
			track_table[i_count].Elevation:=0;
			track_table[i_count].FeedIndexer:=0;
		END_FOR;*)
END_IF

IF b_not_track AND  b_stop_TOA THEN
		i_start:=1;
		i_end:=1;
		track_table[1].TAIoffset:=0;
		FOR i_count:=1 TO i_total BY 1 DO
			track_table[i_count].TAIoffset:=0;
			track_table[i_count].Azimuth:= 0;
			track_table[i_count].Elevation:=0;
			//track_table[i_count].FeedIndexer:=0;
		END_FOR;
		(*track_table[1].MJD:=0;
		FOR i_count:=1 TO i_total BY 1 DO
			track_table[i_count].MJD:=0;
			track_table[i_count].Azimuth:= 0;
			track_table[i_count].Elevation:=0;
			track_table[i_count].FeedIndexer:=0;
		END_FOR; *)
		b_not_track:=FALSE;
		b_stop_TOA:=FALSE;
END_IF


IF i_start = i_end THEN
	b_on_track_mode:=FALSE;
	b_track_pause:=FALSE;
	b_permit_new_file:=TRUE;
END_IF



IF status_code1='A0160' OR status_code1='A0163' THEN
	drive_code1:='AF';
ELSIF  (status_code1='A0013' OR status_code1='A0012' ) AND axisdata[1].Axis_InAb THEN
	drive_code1:='Ab';
ELSIF  (status_code1='A0013' OR status_code1='A0012' ) AND axisdata[1].Axis_Inbb THEN 
	drive_code1:='bb';	
ELSE
	drive_code1:=status_code1;	
END_IF



IF status_code2='A0160' OR status_code2='A0163'THEN
	drive_code2:='AF';
ELSIF  (status_code2='A0013' OR status_code2='A0012' ) AND axisdata[2].Axis_InAb THEN
	drive_code2:='Ab';
ELSIF  (status_code2='A0013' OR status_code2='A0012' ) AND axisdata[2].Axis_Inbb THEN 
	drive_code2:='bb';	
ELSE
	drive_code2:=status_code2;	
END_IF

IF status_code1 = 'E2004' THEN
	drive_code1:=drive_code2;
END_IF

IF status_code3='A0160' OR status_code3='A0163' OR status_code3='A0161' OR status_code3='A0010' OR status_code3='A0101'THEN
	drive_code3:='AF';
ELSIF ( status_code3='A0013' OR status_code3='A0012' ) AND axisdata[3].Axis_InAb THEN
	drive_code3:='Ab';
ELSIF  (status_code3='A0013' OR status_code3='A0012' ) AND axisdata[3].Axis_Inbb THEN 
	drive_code3:='bb';	
ELSE
	drive_code3:=status_code3;	
END_IF

IF status_code4='A0160' OR status_code4='A0163'THEN
	drive_code4:='AF';
ELSIF  (status_code4='A0013' OR status_code4='A0012' ) AND axisdata[4].Axis_InAb THEN
	drive_code4:='Ab';
ELSIF  (status_code4='A0013' OR status_code4='A0012' ) AND axisdata[4].Axis_Inbb THEN 
	drive_code4:='bb';	
ELSE
	drive_code4:=status_code4;	
END_IF

IF status_code5='A0160' OR status_code5='A0163' THEN
	drive_code5:='AF';
ELSIF  (status_code5='A0013' OR status_code5='A0012' ) AND axisdata[5].Axis_InAb THEN
	drive_code5:='Ab';
ELSIF  (status_code5='A0013' OR status_code5='A0012' ) AND axisdata[5].Axis_Inbb THEN 
	drive_code5:='bb';	
ELSE
	drive_code5:=status_code5;	
END_IF

IF status_code6='A0160' OR status_code6='A0163' THEN
	drive_code6:='AF';
ELSIF  (status_code6='A0013' OR status_code6='A0012' )AND axisdata[6].Axis_InAb THEN
	drive_code6:='Ab';
ELSIF  (status_code6='A0013' OR status_code6='A0012' ) AND axisdata[6].Axis_Inbb THEN 
	drive_code6:='bb';	
ELSE
	drive_code6:=status_code6;	
END_IF

IF status_code1='E8029' OR status_code1='E8030' THEN
	b_limit_az:=TRUE;

ELSE
	b_limit_az:=FALSE;
END_IF

fb_r_az_limit(CLK:=b_limit_az);

IF fb_r_az_limit.Q THEN
	r_vel_az:=0;
	b_scc_vel:=TRUE;
END_IF

IF status_code3='E8029' OR status_code3='E8030' THEN
	b_limit_el:=TRUE;
ELSE
	b_limit_el:=FALSE;
END_IF

fb_r_el_limit(CLK:=b_limit_el);

IF fb_r_el_limit.Q THEN
	r_vel_el:=0;
	b_scc_vel:=TRUE;
END_IF

IF status_code5='E8029' OR status_code5='E8030' THEN
	b_limit_FI:=TRUE;
ELSE
	b_limit_FI:=FALSE;
END_IF

fb_r_FI_limit(CLK:=b_limit_FI);

IF fb_r_FI_limit.Q THEN
	r_vel_FI:=0;
	b_scc_vel:=TRUE;
END_IF



(*<<<<<<<<<<<<<<<<<<<<<<<<<<<<<master_status>>>>>>>>>>>>>>>>>>>>>>>>>>>>>>>>>>>>>>>>>>>>>>>>>>>>>>>*)
master_status.0:=(axisdata[1].Axis_InAb AND axisdata[2].Axis_InAb AND axisdata[3].Axis_InAb);
IF b_remote_on=TRUE THEN
	master_status.1:=0;
ELSE
	master_status.1:=1;
END_IF
IF b_DSdoor_ESTOP THEN
	master_status.2:=1;
ELSE
	master_status.2:=0;
END_IF

	master_status.3:=b_stow_lock;
	master_status.4:=(axisdata[1].Axis_Error OR axisdata[2].Axis_Error OR axisdata[3].Axis_Error);
	master_status.5:=b_stow_pin_limit_unlock;
	master_status.6:=b_stow_pin_limit_lock;
	
IF i_num_stack_left>9500 THEN
		master_status.7:=0;
	ELSE IF i_num_stack_left<1500 THEN
		master_status.7:=1;	
	END_IF
END_IF
	master_status.8:=0;
	master_status.9:=0;
	master_status.10:=0;



(*<<<<<<<<<<<<<<<<<<<<<<<<<<<<status_1>>>>>>>>>>>>>>>>>>>>>>>>>>>>>>>>>>>>>>>>>>>>>>>>>>>>>>>*)
status_1.0:=axisdata[1].Axis_InAb;
status_1.1:=axisdata[1].Axis_Power;
//status_1.1:=1;
status_1.2:=status_1.1;
status_1.3:=b_limit_ccw_az;
status_1.4:=b_limit_cw_az;
status_1.5:=axisdata[1].Axis_Error;
(*<<<<<<<<<<<<<<<<<<<<<<<<<<<<<status_2>>>>>>>>>>>>>>>>>>>>>>>>>>>>>>>>>>>>>>>>>>>>>>>>>>>>>>>*)
status_2.0:=axisdata[2].Axis_InAb;
status_2.1:=axisdata[2].Axis_Power;
//status_2.1:=1;
status_2.2:=status_2.1;
status_2.3:=b_limit_ccw_az;
status_2.4:=b_limit_cw_az;
status_2.5:=axisdata[2].Axis_Error;
(*<<<<<<<<<<<<<<<<<<<<<<<<<<<<<status_3>>>>>>>>>>>>>>>>>>>>>>>>>>>>>>>>>>>>>>>>>>>>>>>>>>>>>>>*)
status_3.0:=axisdata[3].Axis_InAb;
status_3.1:=axisdata[3].Axis_Power;
//status_3.1:=1;
status_3.2:=status_3.1;
status_3.3:=b_limit_ccw_el;
status_3.4:=b_limit_cw_el;
status_3.5:=axisdata[3].Axis_Error;

//axisdata[4].Axis_InAb:=axisdata[3].Axis_InAb;
//axisdata[5].Axis_InAb:=axisdata[3].Axis_InAb;
//axisdata[4].Axis_Power:=axisdata[3].Axis_Power;
//axisdata[5].Axis_Power:=axisdata[3].Axis_Power;

(*<<<<<<<<<<<<<<<<<<<<<<<<<<<<<status_4>>>>>>>>>>>>>>>>>>>>>>>>>>>>>>>>>>>>>>>>>>>>>>>>>>>>>>>*)
status_4.0:=axisdata[3].Axis_InAb;
status_4.1:=axisdata[3].Axis_Power;
//status_4.1:=1;
status_4.2:=status_4.1;
status_4.3:=b_limit_ccw_FI;
status_4.4:=b_limit_cw_FI;
status_4.5:=axisdata[3].Axis_Error;
(*<<<<<<<<<<<<<<<<<<<<<<<<<<<<<status_5>>>>>>>>>>>>>>>>>>>>>>>>>>>>>>>>>>>>>>>>>>>>>>>>>>>>>>>*)
status_5.0:=axisdata[3].Axis_InAb;
status_5.1:=axisdata[3].Axis_Power;
//status_5.1:=1;
status_5.2:=status_5.1;
status_5.3:=b_limit_ccw_FI;
status_5.4:=b_limit_cw_FI;
status_5.5:=axisdata[3].Axis_Error;





reply_count:=reply_count+1;
IF reply_count = 50 THEN	
	reply_count:=0;
END_IF

IF reply_count = 25 THEN 

(*<<<<<<<<<<<<<<<<<<<<<<<<<<<<<concatenate STR_GSTAT>>>>>>>>>>>>>>>>>>>>>>>>>>>>>>>>>>>>>>>>>>>>>>>>>>>>>>>*)
				str_concat[1]:='OTHERSTATUS';
				str_concat[2]:=CONCAT(' ',LREAL_TO_STRING(lr_MJD_current));(*在track——running*)
				str_concat[3]:=CONCAT(' ',LREAL_TO_STRING(r_temp_motor1));(*在track——running*)
				str_concat[4]:=CONCAT(' ',LREAL_TO_STRING(r_temp_motor2));
    			str_concat[5]:=CONCAT(' ',LREAL_TO_STRING(r_temp_motor3));
 				str_concat[6]:=CONCAT(' ',LREAL_TO_STRING(r_temp_motor1));
				str_concat[7]:=CONCAT(' ',LREAL_TO_STRING(r_temp_motor2));	
				str_concat[8]:=CONCAT(' ',drive_code1);
				str_concat[9]:=CONCAT(' ',drive_code2);
				str_concat[10]:=CONCAT(' ',drive_code3);
				str_concat[11]:=CONCAT(' ',drive_code1);
				str_concat[12]:=CONCAT(' ',drive_code2);
				str_Send:='';(*for语句格式*)
				FOR Counter:=1 TO 12 BY 1 DO
					str_Send:=CONCAT(str_Send,str_concat[Counter]);
				END_FOR;

	ELSE				
(*<<<<<<<<<<<<<<<<<<<<<<<<<<<<<concatenate STR_GSTAT>>>>>>>>>>>>>>>>>>>>>>>>>>>>>>>>>>>>>>>>>>>>>>>>>>>>>>>*)
				str_concat[1]:='STATUS';
				str_concat[2]:=CONCAT(' ',LREAL_TO_STRING(lr_MJD_current));(*在track——running*)
				str_concat[3]:=CONCAT(' ',UINT_TO_STRING(i_Start));(*在track——running*)
				str_concat[4]:=CONCAT(' ',UINT_TO_STRING(i_End));(*在track——running*)
				str_concat[5]:=CONCAT(' ',INT_TO_STRING(i_num_stack_left));(*在track——running*)
				str_concat[6]:=CONCAT(' ',LREAL_TO_STRING(r_pos_az));
				str_concat[7]:=CONCAT(' ',LREAL_TO_STRING(r_pos_el));
 				str_concat[8]:=CONCAT(' ',LREAL_TO_STRING(r_pos_FI));
				str_concat[9]:=CONCAT(' ','1');   //MLC状态
    			str_concat[10]:=CONCAT(' ',DWORD_TO_STRING(master_status));
				str_concat[11]:=CONCAT(' ',LREAL_TO_STRING(r_following_1));
				str_concat[12]:=CONCAT(' ',LREAL_TO_STRING(r_following_3));
 				str_concat[13]:=CONCAT(' ',DINT_TO_STRING(r_step_count));
			  //str_concat[13]:=CONCAT(' ',REAL_TO_STRING(r_following_5));
				str_concat[14]:=CONCAT(' ',DWORD_TO_STRING(status_1));
				str_concat[15]:=CONCAT(' ',DWORD_TO_STRING(status_2));
				str_concat[16]:=CONCAT(' ',DWORD_TO_STRING(status_3));
				str_concat[17]:=CONCAT(' ',DWORD_TO_STRING(status_4));
				str_concat[18]:=CONCAT(' ',DWORD_TO_STRING(status_5));	
                str_concat[19]:=CONCAT(' ',LREAL_TO_STRING(r_current_1));
                str_concat[20]:=CONCAT(' ',LREAL_TO_STRING(i_speed_1));
                str_concat[21]:=CONCAT(' ',LREAL_TO_STRING(r_current_2));	
                str_concat[22]:=CONCAT(' ',LREAL_TO_STRING(i_speed_2));
                str_concat[23]:=CONCAT(' ',LREAL_TO_STRING(r_current_3));	
				str_concat[24]:=CONCAT(' ',LREAL_TO_STRING(i_speed_3));
				str_concat[25]:=CONCAT(' ',LREAL_TO_STRING(r_current_4));
				str_concat[26]:=CONCAT(' ',LREAL_TO_STRING(i_speed_4));
				str_concat[27]:=CONCAT(' ',LREAL_TO_STRING(r_current_5));
				str_concat[28]:=CONCAT(' ',LREAL_TO_STRING(i_speed_5));
				str_Send:='';(*for语句格式*)
				FOR Counter:=1 TO 28 BY 1 DO
					str_Send:=CONCAT(str_Send,str_concat[Counter]);
				END_FOR;
(*<<<<<<<<<<<<<<<<<<<<<<<<<<<if TCP is wrong,reset the TCP serve>>>>>>>>>>>>>>>>>>>>>>>>>>>>*)
END_IF				
				
				
(*<<<<<<<<<<<<<<<<<<<<<<<<<<<if TCP is wrong,reset the TCP serve>>>>>>>>>>>>>>>>>>>>>>>>>>>>*)
IF TCPConnection.Error=TRUE OR TCPRecv.Error=TRUE OR TCPSend.Error=TRUE THEN
	b_Server_Enable:=FALSE;
	b_Recv_enable:=FALSE;
	b_Send_enable:=FALSE;
ELSE
	b_Server_Enable:=TRUE;
END_IF

IF b_Connection_done = TRUE THEN
	i_counter_tcp := i_counter_tcp + 1;
END_IF;

(*
IF i_counter_tcp>2000 THEN
	B_TCP_close := TRUE;
	b_scc_enable_off := TRUE;
	b_scc_enable_on := FALSE;
	i_counter_tcp :=0;
ELSE
	B_TCP_close:= FALSE;
END_IF;
*)

P_TCP_with_SCC.Async_TCP();
P_TCP_with_SCC.A_RECV();
P_TCP_with_SCC.A_SEND();
(*<<<<<<<<<<<<<<<<<<<<<<<<<<<if TCP server is connected,a cycle is executed>>>>>>>>>>>>>>>>>>>>>>>>>>>>>>>>>>>>>>>>>>>>>*)
IF b_Connection_done=TRUE THEN
	IF  b_receiving=FALSE AND b_commanding=FALSE AND b_sending=FALSE AND b_Recv_enable=FALSE THEN
		b_Recv_enable:=TRUE;(*open recieve fuction*)
		P_TCP_with_SCC.A_RECV();
		b_receiving:=TRUE;
	END_IF;
(*<<<<<<<<<<<<<<<<<<<<<<<<<<<recieveing message>>>>>>>>>>>>>>>>>>>>>>>>>>>>>>>>>>>>>>>>>>>>>>>>>*)
	IF b_Recv_done=TRUE AND b_receiving=TRUE AND b_commanding=FALSE AND b_sending=FALSE THEN
		str_MSG_Received:=CONCAT(str_MSG_Received,LEFT(str_Recv,UDINT_TO_INT(di_ReceivedBytes)));
		fb_msg_receive(str_Message:=str_MSG_Received);
		str_MSG_Received:='';
		b_Recv_enable:=FALSE;
		P_TCP_with_SCC.A_RECV();
		b_receiving:=FALSE;
		b_commanding:=TRUE;
		i_counter_tcp :=0;
	END_IF
(*<<<<<<<<<<<<<<<<<<<<<<<<<<<<<<<<operating function>>>>>>>>>>>>>>>>>>>>>>>>>>>>>>>>>>>>>>>>>>>>>*)
	IF b_receiving=FALSE AND b_commanding=TRUE AND b_sending=FALSE THEN
(*<<<<<<<<<<<<<<<<<<<<<<<<<<<<<ENABLE>>>>>>>>>>>>>>>>>>>>>>>>>>>>>>>>>>>>>>>>>>>>>>>>>>>>>>>*)
		IF fb_msg_receive.Key='ENABLE'  THEN
			IF fb_msg_receive.P_value[1]='ON' THEN
				IF AXISDATA[1].Axis_InAb AND AXISDATA[3].Axis_InAb  THEN(*whether or not Power on*)
					b_off_write:=FALSE;
					b_on_write:=TRUE;
					b_SCC_enable_on:=TRUE;
					b_SCC_enable_off:=FALSE;
					IF b_remote_on THEN
					i_receive_cmd:=i_receive_cmd+1;
					i_excute_cmd:=i_excute_cmd+1;
					last_command:='05';
					END_IF
					str_Send:=F_RPL_1('',str_Send);
					b_commanding:=FALSE;
					b_sending:=TRUE;
				ELSE
					str_Send:=F_RPL_1('',str_Send);
					b_commanding:=FALSE;
					b_sending:=TRUE;
				END_IF;
			ELSIF fb_msg_receive.P_value[1]='OFF' THEN
					
					IF b_scc_vel1_temp THEN
					b_start_adjust_vel:=FALSE;
					b_start_adjust_vel_temp:=FALSE;
					r_vel_az:=0;
					r_vel_el:=0;
					b_scc_vel:=TRUE;
					P_TCP_with_SCC.A_SCC_GOTO();
					vel_stop_ton(IN := b_scc_vel, PT:= T#3S);
					vel_stop_ton.ET;
					IF vel_stop_ton.Q THEN
						b_scc_vel1_temp:=FALSE;
					b_on_write:=FALSE;
					b_off_write:=TRUE;
					b_scc_vel:=FALSE;
					b_scc_enable_off:=TRUE;
					b_SCC_enable_on:=FALSE;
					b_scc_goto:=FALSE;
					b_active_AZ:=FALSE;
					b_active_EL:=FALSE;
					b_active_FI:=FALSE;
					b_goto_Az_done:=FALSE;
					b_goto_EL_done:=FALSE;
					b_goto_FI_done:=FALSE;
					b_SCC_STOP:=FALSE;
					b_stop_act_az:=FALSE;
					b_stop_act_el:=FALSE;
					b_stop_act_FI:=FALSE;
					b_stop1_done:=FALSE;
					b_stop3_done:=FALSE;
					b_stop5_done:=FALSE;
					b_scc_maintain:=FALSE;
					b_scc_stow:=FALSE;
					b_write_az:=FALSE;
					b_write_el:=FALSE;
					b_write_FI:=FALSE;
					b_write_az_done:=FALSE;
					b_write_el_done:=FALSE;
					b_write_FI_done:=FALSE;
					b_open_channel_az:=FALSE;
					b_open_channel_el:=FALSE;
					b_open_channel_FI:=FALSE;
					b_open_channel_az_done:=FALSE;
					b_open_channel_el_done:=FALSE;
					b_open_channel_FI_done:=FALSE;
					b_move_0_done:=FALSE;
					b_move_20_done:=FALSE;
					b_lock_off:=FALSE;
					b_Track_Pause:=FALSE;
					b_track_on:=FALSE;
					b_on_track_mode:=FALSE;
					b_track_on_first:=FALSE;
					B_encoder_home_d1:=FALSE;
					B_encoder_home_d5:=FALSE;
					b_home_d1:=FALSE;
					b_home_d5:=FALSE;
					b_stop_TOA:=FALSE;
					b_move_to_start1:=FALSE;
					b_move_to_start5:=FALSE;
					b_in_positionMode:=FALSE;
					i_adjust_count:=0;
					b_first_pos_done:=FALSE;
					b_second_pos_done:=FALSE;
					b_3rd_pos_done:=FALSE;
					b_4th_pos_done:=FALSE;
					b_5th_pos_done:=FALSE;
					b_6th_pos_done:=FALSE;
					b_7th_pos_done:=FALSE;
					b_8th_pos_done:=FALSE;
					b_9th_pos_done:=FALSE;
					b_10th_pos_done:=FALSE;
					adjust_delay:=FALSE;
					i_closeloop_count:=0;
					END_IF		
					END_IF
					b_start_adjust_vel:=FALSE;
					b_start_adjust_vel_temp:=FALSE;
					b_scc_vel1_temp:=FALSE;
					b_on_write:=FALSE;
					b_off_write:=TRUE;
					b_scc_vel:=FALSE;
					b_scc_enable_off:=TRUE;
					b_SCC_enable_on:=FALSE;
					b_scc_goto:=FALSE;
					b_active_AZ:=FALSE;
					b_active_EL:=FALSE;
					b_active_FI:=FALSE;
					b_goto_Az_done:=FALSE;
					b_goto_EL_done:=FALSE;
					b_goto_FI_done:=FALSE;
					b_SCC_STOP:=FALSE;
					b_stop_act_az:=FALSE;
					b_stop_act_el:=FALSE;
					b_stop_act_FI:=FALSE;
					b_stop1_done:=FALSE;
					b_stop3_done:=FALSE;
					b_stop5_done:=FALSE;
					b_scc_maintain:=FALSE;
					b_scc_stow:=FALSE;
					b_write_az:=FALSE;
					b_write_el:=FALSE;
					b_write_FI:=FALSE;
					b_write_az_done:=FALSE;
					b_write_el_done:=FALSE;
					b_write_FI_done:=FALSE;
					b_open_channel_az:=FALSE;
					b_open_channel_el:=FALSE;
					b_open_channel_FI:=FALSE;
					b_open_channel_az_done:=FALSE;
					b_open_channel_el_done:=FALSE;
					b_open_channel_FI_done:=FALSE;
					b_move_0_done:=FALSE;
					b_move_20_done:=FALSE;
					b_lock_off:=FALSE;
					b_Track_Pause:=FALSE;
					b_track_on:=FALSE;
					b_on_track_mode:=FALSE;
					b_track_on_first:=FALSE;
					B_encoder_home_d1:=FALSE;
					B_encoder_home_d5:=FALSE;
					b_home_d1:=FALSE;
					b_home_d5:=FALSE;
					b_stop_TOA:=FALSE;
					b_move_to_start1:=FALSE;
					b_move_to_start5:=FALSE;
					b_in_positionMode:=FALSE;
					i_adjust_count:=0;
					b_first_pos_done:=FALSE;
					b_second_pos_done:=FALSE;
					b_3rd_pos_done:=FALSE;
					b_4th_pos_done:=FALSE;
					b_5th_pos_done:=FALSE;
					b_6th_pos_done:=FALSE;
					b_7th_pos_done:=FALSE;
					b_8th_pos_done:=FALSE;
					b_9th_pos_done:=FALSE;
					b_10th_pos_done:=FALSE;
					b_SCC_STOP:=FALSE;
					adjust_delay:=FALSE;
					i_closeloop_count:=0;
					lockstand:=TRUE;
					V_LastSpeed:=0;
					V_LastOutput:=0;
					dIntegralSpeed:= 0;	
					V_command_EL:=0;
					b_start_cyclicvel:=FALSE;
					b_write_el_vel:=FALSE;	
					b_step_running:=0;
					b_step_running_az:=0;
					b_step_running_el:=0;
					r_step_count:=0;
					r_step_count_temp:=0;
					b_offset_running:=0;
					r_offset_count_temp:=0;
					r_offset_count:=0;	
					r_offset_az:=0;
					r_offset_el:=0;
					V_LastOutput:=0;
					V_command_EL:=0;
					Pos_EL_error:=0;
					r_test_offset_el:=0;
					r_test_offset_az:=0;
					dIntegralSpeed:=0;
					m_dLastIntegral:=0;
					r_Integral_thistime:=0;
					r_el_offset_abs:=0;
					IF b_remote_on THEN
					i_receive_cmd:=i_receive_cmd+1;
					i_excute_cmd:=i_excute_cmd+1;
					last_command:='06';
					END_IF
				    str_Send:=F_RPL_1('',str_Send);
					b_commanding:=FALSE;
					b_sending:=TRUE;
			ELSE
				   	str_Send:=F_RPL_1('',str_Send);
					b_commanding:=FALSE;
					b_sending:=TRUE;
			END_IF;
(*<<<<<<<<<<<<<<<<<<<<<<<<<<<<<<<<<<<<<<ESTOP>>>>>>>>>>>>>>>>>>>>>>>>>>>>>>>>>>>>>>>>>>>>>>>*)
		ELSIF	fb_msg_receive.Key ='ESTOP'  AND b_remote_on=TRUE THEN
			b_power_Az :=FALSE;
			b_power_el:=FALSE;
			b_power_FI:=FALSE;
	     	str_Send:=F_RPL_1('',str_Send);
					b_commanding:=FALSE;
					b_sending:=TRUE;

(*<<<<<<<<<<<<<<<<<<<<<<<<<<<<<GOTO>>>>>>>>>>>>>>>>>>>>>>>>>>>>>>>>>>>>>>>>*)
		ELSIF fb_msg_receive.Key='GOTO'  THEN
			r_EL_current_when_goto_cmd:=r_pos_el;
			T_count_goto:=0.0;
			Pos_EL_Aim:=r_pos_el;
			r_goto_az_I:=STRING_TO_REAL(fb_msg_receive.P_value[1]);(*input value of GOTO*)
            r_goto_el_I:=STRING_TO_REAL(fb_msg_receive.P_value[2]);
            r_goto_FI_I:=STRING_TO_REAL(fb_msg_receive.P_value[3]);
				IF (-270.01<r_goto_az_I)AND(r_goto_az_I<270.01)AND(14.9<r_goto_el_I)AND(r_goto_el_I<=90)AND(-0.01<r_goto_FI_I)AND(r_goto_FI_I<180.01)THEN
					r_goto_az:=r_goto_az_I-r_pos_az_v;
					vel_move_az_1:=vel_move_az;
						acc_mov_az:=0.08;
						dcc_mov_az:=0.08;				
					b_scc_vel1_temp:=FALSE;
					b_start_adjust_vel:=FALSE;
					r_p0:=ML_Base.AxisData[11].rActualPosition_i;
					r_p1:=Encoder_to_motor(r_goto_el_I);
					r_p2:=Encoder_to_motor(r_p0);
					r_goto_el_abs:=Encoder_to_motor(r_goto_el_I);
					r_goto_el:=Encoder_to_motor(r_goto_el_I)-Encoder_to_motor(ML_Base.AxisData[11].rActualPosition_i);
					r_goto_FI:=r_goto_FI_I-r_pos_FI_v+90;
					b_first_pos_done:=FALSE;
					b_second_pos_done:=FALSE;
					b_3rd_pos_done:=FALSE;
					b_4th_pos_done:=FALSE;
					b_5th_pos_done:=FALSE;
					b_6th_pos_done:=FALSE;
					b_7th_pos_done:=FALSE;
					b_8th_pos_done:=FALSE;
					b_9th_pos_done:=FALSE;
					b_10th_pos_done:=FALSE;
					i_adjust_count:=0;
					adjust_delay:=FALSE;
					i_closeloop_count:=0;					
					b_SCC_STOP:=FALSE;
					b_scc_goto:=TRUE;
					b_start_goto_az_tcp:=TRUE;
					b_step_running_az:=1;
					b_step_running_el:=1;
					r_step_count_temp:=r_step_count_temp+1;
					b_in_positionMode:=TRUE;	
					IF b_remote_on THEN
					i_receive_cmd:=i_receive_cmd+1;
					i_excute_cmd:=i_excute_cmd+1;
					last_command:='02';
					END_IF
					str_Send:=F_RPL_1('',str_Send);
					b_commanding:=FALSE;
					b_sending:=TRUE;
				ELSE
					b_scc_goto:=FALSE;
					b_start_goto_az_tcp:=FALSE;
					str_Send:=F_RPL_1('',str_Send);
					b_commanding:=FALSE;
					b_sending:=TRUE;
				END_IF
(*<<<<<<<<<<<<<<<<<<<<<<<<<<<<<SETSPEED>>>>>>>>>>>>>>>>>>>>>>>>>>>>>>>>>>>>>>>>*)
		ELSIF fb_msg_receive.Key='SETSPEED'  THEN
			vel_move_az:=STRING_TO_REAL(fb_msg_receive.P_value[1])/6;
            vel_move_el:=STRING_TO_REAL(fb_msg_receive.P_value[2])/6;
            vel_move_FI:=STRING_TO_REAL(fb_msg_receive.P_value[3])/6;
			IF b_remote_on THEN
			i_receive_cmd:=i_receive_cmd+1;
			i_excute_cmd:=i_excute_cmd+1;
			last_command:='09';
			END_IF
				IF (vel_move_az>0.5)OR(vel_move_el>0.167)OR(vel_move_FI>0.334)THEN
					IF vel_move_az>0.5 THEN
						vel_move_az:=0.5;
					END_IF
					IF vel_move_el>0.167 THEN
						vel_move_el:=0.167;
					END_IF
					IF vel_move_FI>0.334 THEN
						vel_move_FI:=0.334;
					END_IF	
								
					str_Send:=F_RPL_1('',str_Send);
					b_commanding:=FALSE;
					b_sending:=TRUE;
				ELSE
					str_Send:=F_RPL_1('',str_Send);
					b_commanding:=FALSE;
					b_sending:=TRUE;
				END_IF				
				
				
(*<<<<<<<<<<<<<<<<<<<<<<<<<<<<<VEL>>>>>>>>>>>>>>>>>>>>>>>>>>>>>>>>>>>>>>>>*)
		ELSIF fb_msg_receive.Key='VEL' THEN
			b_scc_goto:=FALSE;
			b_scc_vel:=FALSE;
			b_SCC_STOP:=FALSE;
			b_track_on:=FALSE;
			V_command_EL:=0;
			V_LastSpeed:=0;
			V_LastOutput:=0;
			dIntegralSpeed:= 0;	
			b_start_cyclicvel:=FALSE;
			b_write_el_vel:=FALSE;
			b_start_adjust_vel_temp:=FALSE;
			b_start_adjust_vel:=FALSE;
			r_vel_az:=STRING_TO_REAL(fb_msg_receive.P_value[1])/6;
            r_vel_el:=STRING_TO_REAL(fb_msg_receive.P_value[2])/6;
			r_command_vel:=r_vel_el*6;
            r_vel_FI:=STRING_TO_REAL(fb_msg_receive.P_value[3])/6;
			IF b_remote_on_run=FALSE THEN
					str_Send:=F_RPL_1('',str_Send);
					b_commanding:=FALSE;
					b_sending:=TRUE;
			ELSE
				IF (-0.51<r_vel_az)AND(r_vel_az<0.51)AND(-0.17<r_vel_el)AND(r_vel_el<0.17)AND(-0.334<r_vel_FI)AND(r_vel_FI<0.334)THEN
					IF r_pos_az_v>265 AND r_vel_az>0.083 THEN
						r_vel_az:=0.083;
					END_IF
					
					IF r_pos_az_v<-265 AND r_vel_az<-0.083 THEN
						r_vel_az:=-0.083;
					END_IF
					
					IF r_pos_el_v>88 AND r_vel_el>0.1 THEN
						r_vel_el:=0.05;
					END_IF
					
					IF r_pos_el_v<20 AND r_vel_el<-0.1 THEN
						r_vel_el:=-0.05;
					END_IF

					IF r_pos_FI_v>265 AND r_vel_FI>0.083 THEN
						r_vel_FI:=0.083;
					END_IF
					
					IF r_pos_FI_v<95 AND r_vel_FI<-0.083 THEN
						r_vel_FI:=-0.083;
					END_IF
					r_vel_el:=r_vel_el*11976;//*7.5;
//					r_vel_el:=r_vel_el*12100;//*7.5;
					b_scc_vel:=TRUE;
					str_Send:=F_RPL_1('',str_Send);
					b_commanding:=FALSE;
					b_sending:=TRUE;
				ELSE
					b_scc_vel:=FALSE;
				    str_Send:=F_RPL_1('',str_Send);
					b_commanding:=FALSE;
					b_sending:=TRUE;
				END_IF
			END_IF			
			
(*<<<<<<<<<<<<<<<<<<<<<<<<<<<<<<<<<<<<<<POWER>>>>>>>>>>>>>>>>>>>>>>>>>>>>>>>>>>>>>>>>>>>>>>>*)
		ELSIF fb_msg_receive.Key ='PWR'  THEN
				lockstand:=TRUE;
			IF fb_msg_receive.P_value[1]='ON' THEN
				b_power_on:=FALSE;
				IF axisdata[1].Axis_InAb = 0 THEN
				b_Scc_PWR_on:=FALSE;
				b_Scc_PWR_on:=TRUE;
				b_Scc_PWR_off:=FALSE;
				END_IF;
					str_Send:=F_RPL_1('',str_Send);
					b_commanding:=FALSE;
					b_sending:=TRUE;
			ELSIF fb_msg_receive.P_value[1]='OFF' THEN
				IF b_track_on=FALSE THEN
					b_Scc_PWR_on:=FALSE;
					b_Scc_PWR_off:=TRUE;
					b_scc_goto:=FALSE;
					b_active_AZ:=FALSE;
					b_active_EL:=FALSE;
					b_scc_vel:=FALSE;
					b_active_FI:=FALSE;
					b_goto_Az_done:=FALSE;
					b_goto_EL_done:=FALSE;
					b_goto_FI_done:=FALSE;
					b_SCC_STOP:=FALSE;
					b_stop_act_az:=FALSE;
					b_stop_act_el:=FALSE;
					b_stop_act_FI:=FALSE;
					b_stop1_done:=FALSE;
					b_stop3_done:=FALSE;
					b_stop5_done:=FALSE;
					b_scc_maintain:=FALSE;
					b_scc_stow:=FALSE;
					b_write_az:=FALSE;
					b_write_el:=FALSE;
					b_write_FI:=FALSE;
					b_write_az_done:=FALSE;
					b_write_el_done:=FALSE;
					b_write_FI_done:=FALSE;
					b_open_channel_az:=FALSE;
					b_open_channel_el:=FALSE;
					b_open_channel_FI:=FALSE;
					b_open_channel_az_done:=FALSE;
					b_open_channel_el_done:=FALSE;
					b_open_channel_FI_done:=FALSE;
					b_move_0_done:=FALSE;
					b_move_20_done:=FALSE;
					b_lock_off:=FALSE;
					str_Send:=F_RPL_1('',str_Send);
					b_commanding:=FALSE;
					b_sending:=TRUE;
				ELSE
					str_Send:=F_RPL_1('',str_Send);
					b_commanding:=FALSE;
					b_sending:=TRUE;
				END_IF
			ELSE
				   	str_Send:=F_RPL_1('',str_Send);
					b_commanding:=FALSE;
					b_sending:=TRUE;
			END_IF
(*<<<<<<<<<<<<<<<<<<<<<<<<<<<<<<<<<<<<<<STOP>>>>>>>>>>>>>>>>>>>>>>>>>>>>>>>>>>>>>>>>>>>>>>>*)
		ELSIF fb_msg_receive.Key ='STOP' THEN
		
				IF b_track_on=TRUE THEN
					b_stop_TOA:=TRUE;				
				ELSE
					b_on_track_mode:=FALSE;
					b_track_on_first:=FALSE;
					i_start:=1;
					i_end:=1;
					b_Track_Pause:=FALSE;
					track_table[1].TAIoffset:=0;
					FOR i_count:=1 TO i_total BY 1 DO
					track_table[i_count].TAIoffset:=0;
					track_table[i_count].Azimuth:= 0;
					track_table[i_count].Elevation:=0;
					//track_table[i_count].FeedIndexer:=0;
					//track_table[i_count].Elevation_ori:=0;
					END_FOR;
					(*track_table[1].MJD:=0;
					FOR i_count:=1 TO i_total BY 1 DO
					track_table[i_count].MJD:=0;
					track_table[i_count].Azimuth:= 0;
					track_table[i_count].Elevation:=0;
					track_table[i_count].FeedIndexer:=0;
					track_table[i_count].Elevation_ori:=0;
					END_FOR;*)
					b_SCC_STOP:=TRUE;
					V_LastSpeed:=0;
					V_LastOutput:=0;
					dIntegralSpeed:= 0;	
					V_command_EL:=0;
					b_start_cyclicvel:=FALSE;
					b_write_el_vel:=FALSE;	
					b_Track_Pause:=FALSE;				
				END_IF
				b_SCC_goto:=FALSE;
				IF b_remote_on THEN
				i_receive_cmd:=i_receive_cmd+1;
				i_excute_cmd:=i_excute_cmd+1;
				last_command:='01';
				END_IF
				str_Send:=F_RPL_1('',str_Send);
				b_commanding:=FALSE;
				b_sending:=TRUE;
(*<<<<<<<<<<<<<<<<<<<<<<<<<<<<<<<<<<<<<<STOW>>>>>>>>>>>>>>>>>>>>>>>>>>>>>>>>>>>>>>>>>>>>>>>*)
		ELSIF fb_msg_receive.Key ='STOW' THEN
			b_scc_Unlock:=FALSE;
			IF b_PID_in_el=TRUE THEN
				b_scc_maintain:=FALSE;
				b_scc_stow:=TRUE;
					str_Send:=F_RPL_1('',str_Send);
					b_commanding:=FALSE;
					b_sending:=TRUE;
			ELSE
					str_Send:=F_RPL_1('',str_Send);
					b_commanding:=FALSE;
					b_sending:=TRUE;
			END_IF
(*<<<<<<<<<<<<<<<<<<<<<<<<<<<<<<<<<<<<<<MAINTAIN>>>>>>>>>>>>>>>>>>>>>>>>>>>>>>>>>>>>>>>>>>>>>>>*)
		ELSIF fb_msg_receive.Key ='MAINTAIN'  THEN
		
					b_permit_new_file:=TRUE;		
					str_Send:=F_RPL_1('',str_Send);
					b_commanding:=FALSE;
					b_sending:=TRUE;
			
(*<<<<<<<<<<<<<<<<<<<<<<<<<<<<<<<<<<<<<<HOME>>>>>>>>>>>>>>>>>>>>>>>>>>>>>>>>>>>>>>>>>>>>>>>*)
		ELSIF fb_msg_receive.Key ='HOME' THEN
		
					b_off_write:=FALSE;	
				    b_SCC_enable_off:=FALSE;
					IF b_remote_on THEN	
					i_receive_cmd:=i_receive_cmd+1;
					i_excute_cmd:=i_excute_cmd+1;
					last_command:='08';
					END_IF
			IF b_encoder_ok_az = FALSE THEN 
				B_encoder_home_d1:=TRUE;  
			END_IF
			
			IF b_encoder_ok_FI = FALSE THEN 
				B_encoder_home_d5:=TRUE;
			END_IF			
					str_Send:=F_RPL_1('',str_Send);
					b_commanding:=FALSE;
					b_sending:=TRUE;
				
(*<<<<<<<<<<<<<<<<<<<<<<<<<<<<<<<<<<<<<<unlock>>>>>>>>>>>>>>>>>>>>>>>>>>>>>>>>>>>>>>>>>>>>>>>*)
		ELSIF fb_msg_receive.Key ='UNLOCK' AND b_remote_on=TRUE THEN
			IF b_stow_pin_limit_unlock=TRUE  THEN
				b_scc_stow:=FALSE;
				b_scc_maintain:=FALSE;
				b_scc_Unlock:=TRUE;
					str_Send:=F_RPL_1('',str_Send);
					b_commanding:=FALSE;
					b_sending:=TRUE;
			ELSE
					str_Send:=F_RPL_1('',str_Send);
					b_commanding:=FALSE;
					b_sending:=TRUE;
			END_IF
(*<<<<<<<<<<<<<<<<<<<<<<<<<<<<<TRACK>>>>>>>>>>>>>>>>>>>>>>>>>>>>>>>>>>>>>>>>>>>>>>>>>>>>>>>*)
		ELSIF fb_msg_receive.Key='TRACK'  THEN
				b_scc_goto:=FALSE;
			IF fb_msg_receive.P_value[1]='ON' THEN
				IF b_remote_on_run=TRUE  THEN
					IF i_end<>i_START THEN
						b_track_on:=TRUE;
						b_stop_TOA:=FALSE;
						b_not_track:=FALSE;
						b_track_on_first:=TRUE;
						b_on_track_mode:=TRUE;
					b_Track_Pause:=FALSE;
					IF b_remote_on THEN
					i_receive_cmd:=i_receive_cmd+1;
					i_excute_cmd:=i_excute_cmd+1;
					last_command:='03';
					END_IF
					str_Send:=F_RPL_1('',str_Send);
					b_commanding:=FALSE;
					b_sending:=TRUE;
					ELSE
					str_Send:=F_RPL_1('',str_Send);
					b_commanding:=FALSE;
					b_sending:=TRUE;
					END_IF
				ELSE
					str_Send:=F_RPL_1('',str_Send);
					b_commanding:=FALSE;
					b_sending:=TRUE;
				END_IF
			ELSIF fb_msg_receive.P_value[1]='OFF' THEN
				
					b_track_on:=FALSE;
					b_on_track_mode:=FALSE;
					b_track_on_first:=FALSE;
					i_start:=1;
					i_end:=1;
					b_Track_Pause:=FALSE;
					track_table[1].TAIoffset:=0;
					FOR i_count:=1 TO i_total BY 1 DO
					track_table[i_count].TAIoffset:=0;
					track_table[i_count].Azimuth:= 0;
					track_table[i_count].Elevation:=0;
					//track_table[i_count].FeedIndexer:=0;
					//track_table[i_count].Elevation_ori:=0;
					END_FOR;
				(*	track_table[1].MJD:=0;
					FOR i_count:=1 TO i_total BY 1 DO
					track_table[i_count].MJD:=0;
					track_table[i_count].Azimuth:= 0;
					track_table[i_count].Elevation:=0;
					track_table[i_count].FeedIndexer:=0;
					track_table[i_count].Elevation_ori:=0;
					END_FOR; *)
//					b_SCC_STOP:=TRUE;
					b_Track_Pause:=FALSE;				
					b_SCC_goto:=FALSE;
			
(*					
				IF i_start<>i_end THEN
				
					i_pause_temp:=i_start;
					t_difference:=(entry_buffer1[F_I_number(i_start)].MJD-entry_buffer1[F_I_number(i_start-1)].MJD)*86400;
					r_a0:=entry_buffer1[F_I_number(i_start)].Azimuth-entry_buffer1[F_I_number(i_start-1)].Azimuth;
					v_a0:=r_a0/t_difference;
					a_a0:=-v_a0/3;
					i_stop:=ABS(REAL_TO_INT(2.0/t_difference));
					i_stop_1:=ABS(REAL_TO_INT(5/t_difference));

			
					r_az_pause_pos1:=r_pos_az_v + v_a0*0.5 + 0.5*a_a0*0.5*0.5;
					r_az_pause_pos2:=r_pos_az_v + v_a0*1 + 0.5*a_a0*1*1;
					r_az_pause_pos3:=r_pos_az_v + v_a0*1.5 + 0.5*a_a0*1.5*1.5;
					r_az_pause_pos4:=r_pos_az_v + v_a0*2 + 0.5*a_a0*2*2;
					r_az_pause_pos5:=r_pos_az_v + v_a0*2.5 + 0.5*a_a0*2.5*2.5;
					r_az_pause_pos6:=r_pos_az_v + v_a0*3 + 0.5*a_a0*3*3;
					r_az_pause_pos7:=r_pos_az_v + v_a0*3 + 0.5*a_a0*3*3;
					
					entry_buffer1[F_I_number(i_start+1)].Azimuth:=r_az_pause_pos1;
					entry_buffer1[F_I_number(i_start+2)].Azimuth:=r_az_pause_pos2;
					entry_buffer1[F_I_number(i_start+3)].Azimuth:=r_az_pause_pos3;
					entry_buffer1[F_I_number(i_start+4)].Azimuth:=r_az_pause_pos4;
					entry_buffer1[F_I_number(i_start+5)].Azimuth:=r_az_pause_pos5;
					entry_buffer1[F_I_number(i_start+6)].Azimuth:=r_az_pause_pos6;
					entry_buffer1[F_I_number(i_start+7)].Azimuth:=r_az_pause_pos7;
					entry_buffer1[F_I_number(i_start+8)].Azimuth:=r_az_pause_pos7;
					entry_buffer1[F_I_number(i_start+9)].Azimuth:=r_az_pause_pos7;
					entry_buffer1[F_I_number(i_start+10)].Azimuth:=r_az_pause_pos7;
										
					entry_buffer1[F_I_number(i_start+1)].MJD:=lr_MJD_current+0.0000058;
					entry_buffer1[F_I_number(i_start+2)].MJD:=lr_MJD_current+0.0000058*2;
					entry_buffer1[F_I_number(i_start+3)].MJD:=lr_MJD_current+0.0000058*3;
					entry_buffer1[F_I_number(i_start+4)].MJD:=lr_MJD_current+0.0000058*4;
					entry_buffer1[F_I_number(i_start+5)].MJD:=lr_MJD_current+0.0000058*5;
					entry_buffer1[F_I_number(i_start+6)].MJD:=lr_MJD_current+0.0000058*6;	
					entry_buffer1[F_I_number(i_start+7)].MJD:=lr_MJD_current+0.0000058*7;	
					entry_buffer1[F_I_number(i_start+8)].MJD:=lr_MJD_current+0.0000058*8;	
					entry_buffer1[F_I_number(i_start+9)].MJD:=lr_MJD_current+0.0000058*9;	
					entry_buffer1[F_I_number(i_start+10)].MJD:=lr_MJD_current+0.0000058*10;	
			END_IF			
										
                    IF b_on_track_mode THEN 
						b_Track_Pause:=TRUE;
					END_IF
*)
					b_track_on_first:=FALSE;
						
					str_Send:=F_RPL_1('',str_Send);
					b_commanding:=FALSE;
					b_sending:=TRUE;
			END_IF
(*<<<<<<<<<<<<<<<<<<<<<<<<<<<<<TRKVAL>>>>>>>>>>>>>>>>>>>>>>>>>>>>>>>>>>>>>>>>>>>>>>>>>>>>>>>*)
		ELSIF fb_msg_receive.Key='TRKVAL'  THEN
			IF fb_msg_receive.P_value[1]='OFF' THEN
				i_start:=1;
				i_end:=1;
				b_on_track_mode:=FALSE;
				b_track_on_first:=FALSE;
				b_track_on:=FALSE;
				b_Track_Pause:=FALSE;
				track_table[1].TAIoffset:=0;
				FOR i_count:=1 TO i_total BY 1 DO
					track_table[i_count].TAIoffset:=0;
					track_table[i_count].Azimuth:= 0;
					track_table[i_count].Elevation:=0;
					//track_table[i_count].FeedIndexer:=0;
				END_FOR;
			(*	track_table[1].MJD:=0;
				FOR i_count:=1 TO i_total BY 1 DO
					track_table[i_count].MJD:=0;
					track_table[i_count].Azimuth:= 0;
					track_table[i_count].Elevation:=0;
					track_table[i_count].FeedIndexer:=0;
				END_FOR; *)
					str_Send:=F_RPL_1('',str_Send);
					b_commanding:=FALSE;
					b_sending:=TRUE;
			ELSE
			fb_Trkval(
				str_MJD:=fb_msg_receive.P_value[1],
				str_Azimuth:=fb_msg_receive.P_value[2],
				str_Elevation:=fb_msg_receive.P_value[3],
	        	str_FeedIndexer:=fb_msg_receive.P_value[4]);
				
				b_not_track:=false;	
				b_permit_new_file:=FALSE;
				str_Send:=F_RPL_1('',str_Send);
					b_commanding:=FALSE;
					b_sending:=TRUE;
			END_IF;
(*<<<<<<<<<<<<<<<<<<<<<<<<<<<<<UPDATE of NTP>>>>>>>>>>>>>>>>>>>>>>>>>>>>>>>>>>>>>>>>>>>>>>>>>>>>>>>*)
		ELSIF fb_msg_receive.Key='SNTP' THEN
			IF b_track_on=FALSE THEN
				b_NTP_update_start:=TRUE;
					str_Send:=F_RPL_1('',str_Send);
					b_commanding:=FALSE;
					b_sending:=TRUE;
			ELSE
					str_Send:=F_RPL_1('',str_Send);
					b_commanding:=FALSE;
					b_sending:=TRUE;
			END_IF
(*<<<<<<<<<<<<<<<<<<<<<<<<<<<<<GSTAT>>>>>>>>>>>>>>>>>>>>>>>>>>>>>>>>>>>>>>>>>>>>>>>>>>>>>>>*)
		ELSIF fb_msg_receive.Key='GSTAT' THEN


      		      	str_Send:=F_RPL_1('',str_Send);
					b_commanding:=FALSE;
					b_sending:=TRUE;
(*<<<<<<<<<<<<<<<<<<<<<<<<<<<<<<<<<<<<<<K1STAT>>>>>>>>>>>>>>>>>>>>>>>>>>>>>>>>>>>>>>>>>>>>>>>*)
		ELSIF fb_msg_receive.Key ='K1STAT' THEN
			str_Send:='OK - CECT54_12m_V1.1 006-336-918 -179 359 15 90.1 -179 179 90 0 0 0';
					b_commanding:=FALSE;
					b_sending:=TRUE;
(*<<<<<<<<<<<<<<<<<<<<<<<<<<<<<<<<<<<<<<K2STAT>>>>>>>>>>>>>>>>>>>>>>>>>>>>>>>>>>>>>>>>>>>>>>>*)
		ELSIF fb_msg_receive.Key ='K2STAT' THEN
				str_Send:=F_RPL_1('',str_Send);
					b_commanding:=FALSE;
					b_sending:=TRUE;
(*<<<<<<<<<<<<<<<<<<<<<<<<<<<<<<<<<<<<<<K3STAT>>>>>>>>>>>>>>>>>>>>>>>>>>>>>>>>>>>>>>>>>>>>>>>*)
		ELSIF fb_msg_receive.Key ='K3STAT' THEN
			status_K3.0:=b_estop_dr;
			status_K3.1:=b_estop_az;
			status_K3.2:=b_estop_el;
			status_K3.3:=b_estop_FI;
			status_K3.4:=b_estop_mc;
			str_Send:=CONCAT('OK - ',DWORD_TO_STRING(status_K3));
					b_commanding:=FALSE;
					b_sending:=TRUE;
					
(*<<<<<<<<<<<<<<<<<<<<<<<<<<<<<<<<<<<<<<LOCKSTANDBY>>>>>>>>>>>>>>>>>>>>>>>>>>>>>>>>>>>>>>>>>>>>>>>*)
		ELSIF	fb_msg_receive.Key ='LOCKSTANDBY' THEN
				i_counter_1s:=0;
				b_stow:=FALSE;
				b_power_on:=FALSE;
				b_Scc_PWR_on:=FALSE;
				lockstand:=TRUE;
				b_track_on:=FALSE;	
				b_SCC_enable_on:=FALSE;
				b_SCC_enable_off:=FALSE;	
				b_off_write:=FALSE;	
			  	str_Send:=F_RPL_1('',str_Send);
					b_commanding:=FALSE;
					b_sending:=TRUE;			
(***********************OFFSET*************************)
    	 ELSIF fb_msg_receive.Key='OFFSET' THEN
			i_counter_1s:=0;
			r_offset_az_I:=STRING_TO_REAL(fb_msg_receive.P_value[1]);
            r_offset_el_I:=STRING_TO_REAL(fb_msg_receive.P_value[2]);
			
			IF b_track_on  THEN
				b_offset:=TRUE;
				b_test_offset_start:=TRUE;
				str_Send:=F_RPL_1('',str_Send);;
			ELSE
				b_offset:=FALSE;
				b_test_offset_start:=FALSE;
				str_Send:=F_RPL_1('',str_Send);
			END_IF
					b_commanding:=FALSE;
					b_sending:=TRUE;	
(*新加入的累计偏置，一次只能识别加减一次*)
(*				r_offset_az:=r_offset_az+r_offset_az_I;
				r_offset_el:=r_offset_el+r_offset_el_I;
*)
				r_offset_az:=r_offset_az_I-r_offset_az_old;
				r_offset_el:=r_offset_el_I-r_offset_el_old;
//				r_offset_el_program:=r_offset_el_I;
			IF r_offset_az_I=0 AND r_offset_el_I=0 THEN
				r_offset_az:=-r_offset_az_old;
				r_offset_el:=-r_offset_el_old;
				b_offset_running:=TRUE;
				r_offset_count_temp:=r_offset_count_temp+1;
			END_IF;					
(*<<<<<<<<<<<<<<<<<<<<<<<<<<<<<<<<<<<<<<K4STAT>>>>>>>>>>>>>>>>>>>>>>>>>>>>>>>>>>>>>>>>>>>>>>>*)
		ELSIF fb_msg_receive.Key ='K4STAT' THEN
				str_Send:=F_RPL_1('',str_Send);
					b_commanding:=FALSE;
					b_sending:=TRUE;
(*<<<<<<<<<<<<<<<<<<<<<<<<<<<<<<<<<<<<<K5STAT>>>>>>>>>>>>>>>>>>>>>>>>>>>>>>>>>>>>>>>>>>>>>>>>*)
		ELSIF fb_msg_receive.Key ='K5STAT' THEN
				str_Send:=F_RPL_1('',str_Send);
					b_commanding:=FALSE;
					b_sending:=TRUE;
(*<<<<<<<<<<<<<<<<<<<<<<<<<<<<<<<<<<<<<<VERSION>>>>>>>>>>>>>>>>>>>>>>>>>>>>>>>>>>>>>>>>>>>>>>>*)
		ELSIF fb_msg_receive.Key ='VERSION' THEN
			str_Send:=CONCAT('VERSION=V1.1',' CETC54 27 JUL 2015 Alex');
				
					b_commanding:=FALSE;
					b_sending:=TRUE;
(*<<<<<<<<<<<<<<<<<<<<<<<<<<<<<<<<<<<<<<TSTAT>>>>>>>>>>>>>>>>>>>>>>>>>>>>>>>>>>>>>>>>>>>>>>>*)
		ELSIF fb_msg_receive.Key='TSTAT' THEN
			str_Send:=CONCAT('OK -',CONCAT(' ',INT_TO_STRING(i_num_stack_left)));
 			str_Send:=CONCAT(str_Send,CONCAT(' ',REAL_TO_STRING(r_track_error[1])));
			str_Send:=CONCAT(str_Send,CONCAT(' ',REAL_TO_STRING(r_track_error[2])));
			str_Send:=CONCAT(str_Send,CONCAT(' ',REAL_TO_STRING(r_track_error[3])));
					b_commanding:=FALSE;
					b_sending:=TRUE;
		ELSE
			IF b_remote_on=FALSE THEN
					str_Send:=F_RPL_1('',str_Send);
					b_commanding:=FALSE;
					b_sending:=TRUE;
			ELSE
					str_Send:=F_RPL_1('',str_Send);
					b_commanding:=FALSE;
					b_sending:=TRUE;
			END_IF
		END_IF;
	END_IF;
	

(*<<<<<<<<<<<<<<<<<<<<<<<<<<<<<<<<<<<<<<<<<<<<<<<<<send message>>>>>>>>>>>>>>>>>>>>>>>>>>>>>>>>>>>>>>>>>>>>>>>>>>>>>>>*)
	IF b_receiving=FALSE AND b_commanding=FALSE AND b_sending=TRUE THEN
		b_Send_enable:=TRUE;
		P_TCP_with_SCC.A_SEND();
	END_IF
(*<<<<<<<<<<<<<<<<<<<<<<<<<<<<<<<<<<<<<<<<after message is sent,disable send function>>>>>>>>>>>>>>>>>>>>>>>>>>>>>>>>>>>>> *)
	IF b_Send_done=TRUE AND b_sending=TRUE THEN
		str_Send:='';
		b_Send_enable:=FALSE;
		P_TCP_with_SCC.A_SEND();
		b_sending:=FALSE;
	END_IF;
	
	IF b_Connection_done= TRUE THEN

	i_counter_1s:=i_counter_1s+1;
	IF i_counter_1s=2 THEN
		i_counter_1s:=0;
		str_Send:=F_RPL_1('',str_Send);
		b_send_enable:=TRUE;
		P_TCP_with_SCC.A_SEND();
	END_IF
	IF b_Send_done=TRUE  THEN
		str_Send:='';
		b_send_enable:=FALSE;
		P_TCP_with_SCC.A_SEND();
	END_IF;
END_IF;

(*<<<<<<<<<<<<<<<<<<<<<<<<<<<<<<<<<<<<<<<<<<<<<If not conected,then reset receive and send function>>>>>>>>>>>>>>>>>>>>>>>>>>>>>>>>>>>>>>>>>>>>>>>>>>>>>>>*)
ELSE
	b_receiving:=FALSE;
	b_commanding:=FALSE;
	b_sending:=FALSE;
	b_Recv_enable:=FALSE;
	b_send_enable:=FALSE;
END_IF;		

	
(*if TCP on 4242 is sending message,the TCP sending for blackbox(4343) is not allowed*)
//b_send_blackbox_admin:=NOT(b_Send_enable);
(*<<<<<<<<<<<<<<<<<<<<<the action of TCP command,goto,power and stop>>>>>>>>>>>>>>>>>>>>>>>>>>*)
P_TCP_with_SCC.A_SCC_GOTO();
P_TCP_with_SCC.A_SCC_POWER();
P_TCP_with_SCC.A_SCC_STOP();

ACTION Async_TCP:
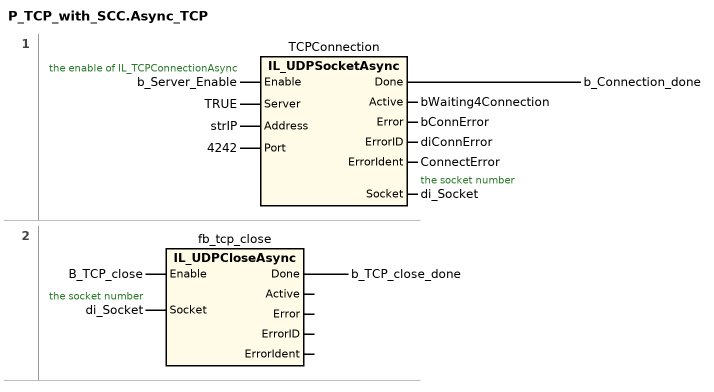
// NETWORK 1
//   b_Server_Enable: the enable of IL_TCPConnectionAsync
//   di_Socket: the socket number
TCPConnection(
    Enable := b_Server_Enable,
    Server := TRUE,
    Address := strIP,
    Port := 4242,
    Active => bWaiting4Connection,
    Error => bConnError,
    ErrorID => diConnError,
    ErrorIdent => ConnectError,
    Socket => di_Socket); // IL_UDPSocketAsync
b_Connection_done := TCPConnection.Done;

// NETWORK 2
//   di_Socket: the socket number
fb_tcp_close(Enable := B_TCP_close, Socket := di_Socket); // IL_UDPCloseAsync
b_TCP_close_done := fb_tcp_close.Done;
END_ACTION

ACTION A_RECV:
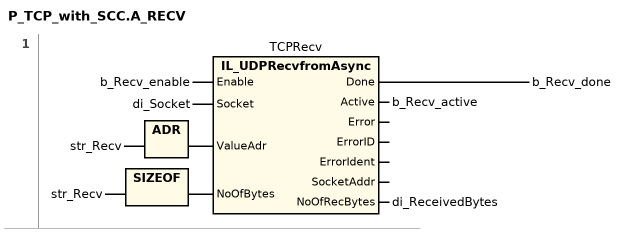
// NETWORK 1
TCPRecv(
    Enable := b_Recv_enable,
    Socket := di_Socket,
    ValueAdr := ADR(str_Recv),
    NoOfBytes := SIZEOF(str_Recv),
    Active => b_Recv_active,
    NoOfRecBytes => di_ReceivedBytes); // IL_UDPRecvfromAsync
b_Recv_done := TCPRecv.Done;
END_ACTION

ACTION A_SCC_GOTO:
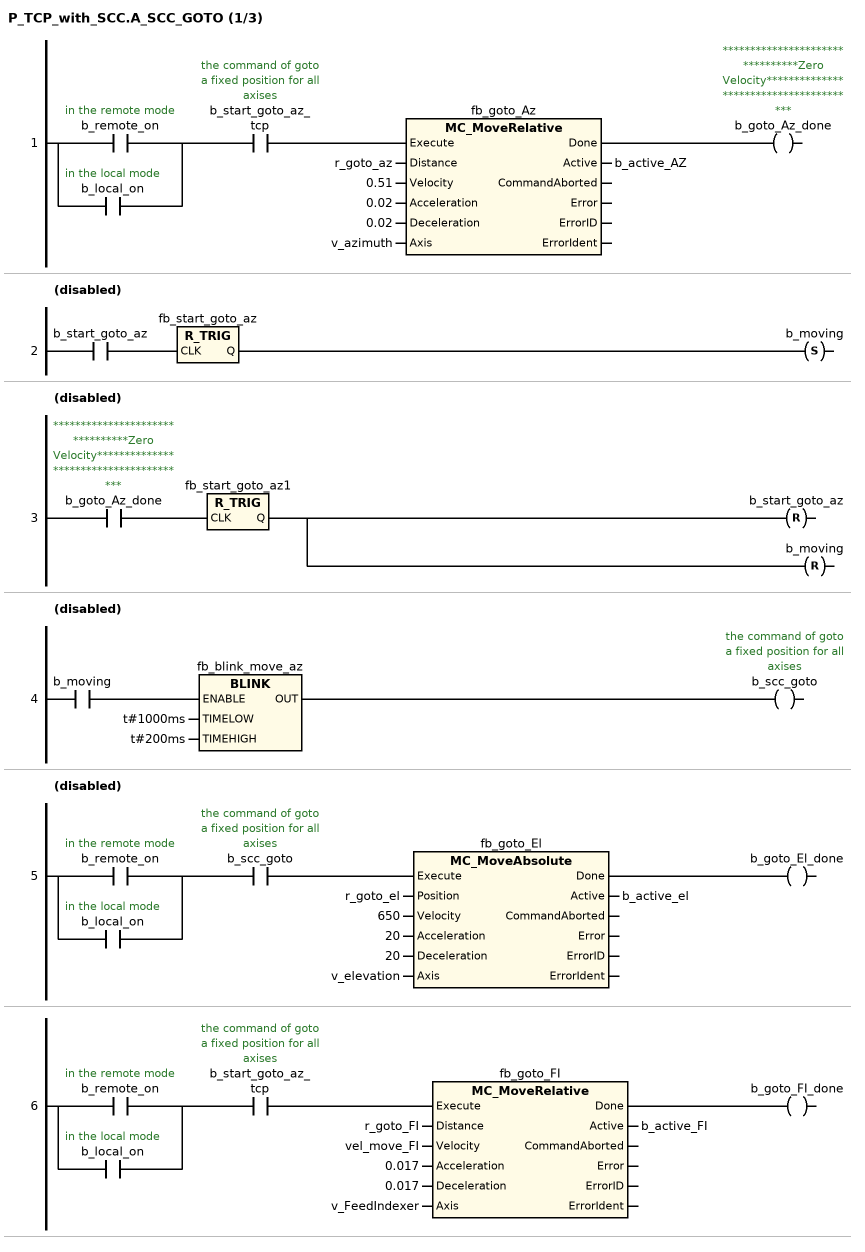
// NETWORK 1
//   b_remote_on: in the remote mode
//   b_local_on: in the local mode
//   b_start_goto_az_tcp: the command of goto a fixed position for all axises
//   r_goto_az: actual value of goto
//   v_azimuth: Virtual axis "v_azimuth" with axis number 7
//   b_goto_Az_done: ********************************Zero Velocity***************************************
fb_goto_Az(
    Execute := (b_remote_on OR b_local_on) AND b_start_goto_az_tcp,
    Distance := r_goto_az,
    Velocity := 0.51,
    Acceleration := 0.02,
    Deceleration := 0.02,
    Axis := v_azimuth,
    Active => b_active_AZ); // MC_MoveRelative
b_goto_Az_done := fb_goto_Az.Done;

// NETWORK 2 (disabled)
// fb_start_goto_az(CLK := b_start_goto_az); // R_TRIG
// b_moving S= fb_start_goto_az.Q;

// NETWORK 3 (disabled)
//   b_goto_Az_done: ********************************Zero Velocity***************************************
// fb_start_goto_az1(CLK := b_goto_Az_done); // R_TRIG
// b_start_goto_az R= fb_start_goto_az1.Q;
// b_moving R= fb_start_goto_az1.Q;

// NETWORK 4 (disabled)
//   b_scc_goto: the command of goto a fixed position for all axises
// fb_blink_move_az(ENABLE := b_moving, TIMELOW := t#1000ms, TIMEHIGH := t#200ms); // BLINK
// b_scc_goto := fb_blink_move_az.OUT;

// NETWORK 5 (disabled)
//   b_remote_on: in the remote mode
//   b_local_on: in the local mode
//   b_scc_goto: the command of goto a fixed position for all axises
//   v_elevation: Virtual axis "v_elevation" with axis number 8
// fb_goto_El(
//     Execute := (b_remote_on OR b_local_on) AND b_scc_goto,
//     Position := r_goto_el,
//     Velocity := 650,
//     Acceleration := 20,
//     Deceleration := 20,
//     Axis := v_elevation,
//     Active => b_active_el); // MC_MoveAbsolute
// b_goto_El_done := fb_goto_El.Done;

// NETWORK 6
//   b_remote_on: in the remote mode
//   b_local_on: in the local mode
//   b_start_goto_az_tcp: the command of goto a fixed position for all axises
//   v_FeedIndexer: Virtual axis "v_polarization" with axis number 9
fb_goto_FI(
    Execute := (b_remote_on OR b_local_on) AND b_start_goto_az_tcp,
    Distance := r_goto_FI,
    Velocity := vel_move_FI,
    Acceleration := 0.017,
    Deceleration := 0.017,
    Axis := v_FeedIndexer,
    Active => b_active_FI); // MC_MoveRelative
b_goto_FI_done := fb_goto_FI.Done;

